FUNCTION_BLOCK FB_Reactor_Set
VAR_IN_OUT
	//stop_reactor_set													: BOOL;
	stop_rs_automode													: BOOL;
	clear_reactor_set_pause												: BOOL;
END_VAR
VAR_INPUT
	r1																	: FB_Reactor;
	
	rs_name																: STRING;
	cycle_mode															: STRING;
//	stop_rs_automode													: BOOL;
	clear_rs_pause														: BOOL;
	open_doors															: BOOL;
	close_doors															: BOOL;
	close_valves														: BOOL;
	retract_clamps														: BOOL;
	extend_clamps														: BOOL;
	
	{attribute 'OPC.UA.DA' := '1'}  				                
	fan_setpoint														: REAL;
	{attribute 'OPC.UA.DA' := '1'}  				                
	{attribute 'OPC.UA.DA.Access' := '1'}  				                
	ti_Cycle_Count														: INT; 
	{attribute 'OPC.UA.DA' := '1'}  				                
	{attribute 'OPC.UA.DA.Access' := '1'}  				                
	ti_Total_Cycle_Count												: DINT; 
	{attribute 'OPC.UA.DA' := '1'}  				                
	{attribute 'OPC.UA.DA.Access' := '1'}  				                
	cycle_stage															: STRING;
    /// <summary>RS_XV08</summary>
	{attribute 'OPC.UA.DA' := '1'}  				                
	steam_bypass_valve													: BOOL;
	/// <summary>XV02</summary>
	{attribute 'OPC.UA.DA' := '1'}  	//mm 11/7 to command valve
	repres_valves														: BOOL;
END_VAR
VAR_OUTPUT
	
	inlet_doors_open													: BOOL;
	inlet_doors_closed													: BOOL;
	outlet_doors_open													: BOOL;
	outlet_doors_closed													: BOOL;

	inlet_clamps_extended												: BOOL;
	inlet_clamps_retracted												: BOOL;
	outlet_clamps_extended												: BOOL;
	outlet_clamps_retracted												: BOOL;
	
	rs_valves_clear														: BOOL;
	adsorption_high_temp_count											: INT;
	desorption_high_temp_count											: INT;
	vacuum_cooling_high_temp_count										: INT;
	sorbent_high_temp													: REAL;
	sorbent_average_temp												: REAL;
	
    /// <summary>Reactor XV02</summary>
	repres_valves_clear													: BOOL;
    /// <summary>RS_XV04</summary>
	dead_air_valve_clear												: BOOL;
    /// <summary>RS_XV05</summary>
	product_iso_valve_clear												: BOOL;
    /// <summary>RS_XV06</summary>
	condensate_valve_clear												: BOOL;
    /// <summary>RS_XV07</summary>
	steam_iso_valve_clear												: BOOL;
    /// <summary>RS_XV08</summary>
	steam_bypass_valve_clear											: BOOL;
	
	/// <summary>RS_LS01</summary>
	{attribute 'OPC.UA.DA' := '1'}  				                
	{attribute 'OPC.UA.DA.Access' := '1'}  				                
	reactor_drain_vessel_lsl									AT %I*	: BOOL;
    /// <summary>RS_LS02</summary>
	{attribute 'OPC.UA.DA' := '1'}  				                
	{attribute 'OPC.UA.DA.Access' := '1'}  				                
	reactor_drain_vessel_lsh									AT %I*	: BOOL;

    /// <summary>RS_FT02</summary>
	{attribute 'OPC.UA.DA' := '1'}  				                
	{attribute 'OPC.UA.DA.Access' := '1'}  				                
	reactor_condensate_flow												: REAL;

	Remaining_Time														: REAL;
	Current_Step														: INT;
	Machine_State														: INT;
	Status																: INT;
	Process_Running														: BOOL;
	Pause_Reactor_Set													: BOOL;
	Reactor_Set_Stopped													: BOOL;
	DoorCycle_Running													: BOOL;
	PositivePressure_Running											: BOOL;
	Repressurization_Running											: BOOL;
	Adsorption_Running													: BOOL;
	Evacuation_Running													: BOOL;
	Desorption_Running													: BOOL;
	Bypass_Running														: BOOL;
	Utility_Error														: BOOL;
	Cancel_Reactor_Set													: BOOL;
	Cancel_All_Reactor_Sets												: BOOL;
	Process_Complete													: BOOL;
	Done																: BOOL;
	
END_VAR
VAR
	eState																: E_MachineState;
	i																	: INT;
	iStatePointer														: INT;
	iLength																: INT;
	iStateMode															: ARRAY[0..9] OF INT;
	stop_reactor_set													: BOOL;
	
	sUtilityError														: STRING;
	sReactorError														: STRING;
	sCancelError														: STRING;
	sRetryError															: STRING;
	sError																: STRING;
	sMessage															: STRING;
	sLeakageAcceptable													: STRING;
	sLeakageUnacceptable												: STRING;

	rAveragePressure													: REAL;
	iCount																: INT;
	iVacuumStatus														: INT;
	iError																: INT;
	
	rTime																: REAL;
	rTime1																: REAL;
	rTime2																: REAL;
	rTime3																: REAL;
	rSP1																: REAL;
	rSP2																: REAL;
	rSP3																: REAL;
	rR1SavedPressure													: REAL;
	rR1Leakage															: REAL;
	rIncrementalMove													: REAL;
	rPosition															: REAL;
	rAverageReactorPres													: REAL;
	rReactorLeakTestStartingPressure									: REAL;
	
	tTime																: TIME;
	
	iStep																: INT;
	i2Step																: INT;
	i3Step																: INT;
	i4Step																: INT;
	i5Step																: INT;
	i6Step																: INT;
	i7Step																: INT;
	i8Step																: INT;
	iStartStep															: INT;
	iStatus																: INT;
	iErrorProcess														: INT;
	iR1Leakage															: INT;
	iCycleCount															: INT;
	iMaxSorbentTempErrorCount											: INT;

	bMultiProcess														: BOOL;
	bEndProcess															: BOOL;
	bSPAdjust															: BOOL;
	bPaused																: BOOL;
	bClearingCycle														: BOOL;
	bDoorCycleDone								        				: BOOL;
	bPositivePressureDone						        				: BOOL;
	bRepressurizationDone												: BOOL;
	bAdsorptionDone														: BOOL;
	bEvacuationDone														: BOOL;
	bDesorptionDone									        			: BOOL;
	bBypassDone									        				: BOOL;
	bPass1																: BOOL;
	bPass2																: BOOL;
	bPass3																: BOOL;
	bPass4																: BOOL;
	bPass5																: BOOL;
	bPass6																: BOOL;
	bPass7																: BOOL;
	bPass8																: BOOL;
	bPass9																: BOOL;
	bPass10																: BOOL;
	
	
	bCondenserKnockoutOn												: BOOL;
	bStop																: BOOL;
	bTimer1																: BOOL;
	bTimer2																: BOOL;
	bTimer3																: BOOL;
	bRunning															: BOOL;
	bDrainError															: BOOL;
	bPumpOn																: BOOL;
	bPumpTimeOut														: BOOL;									
	bDrainResetToLSL													: BOOL;
	bProcessStarted														: BOOL;
	bDesorptionErrorCheck												: BOOL;
	bSafeShutdownOn														: BOOL;
	bInletClampsRetracted												: BOOL;
	bInletClampsExtended												: BOOL;
	bOutletClampsRetracted												: BOOL;
	bOutletClampsExtended												: BOOL;
	bVacuumHolding														: BOOL;
	bCondition21														: BOOL;
	bCondition22														: BOOL;
	bCondition11														: BOOL;
	bCondition12														: BOOL;
	
	rtrigStart															: R_TRIG;
	rtrigPaused															: R_TRIG;
	rtrigIdle															: R_TRIG;
	rtrigDoorCycle														: R_TRIG;
	rtrigPositivePressure												: R_TRIG;
	rtrigRepressurization												: R_TRIG;
	rtrigAdsorption														: R_TRIG;
	rtrigEvacuation														: R_TRIG;
	rtrigDesorption														: R_TRIG;
	rtrigBypass															: R_TRIG;
	rtrigSingleProcessAuto												: R_TRIG;
	rtrigDrainLSHOn														: R_TRIG;
	
	tonTimer1															: TON;
	tonTimer2															: TON;
	tonTimer3															: TON;
	tonPause															: TON;
	tonDrain															: TON;
	rtrigCondensateValveOff_DrainOff									: R_TRIG;
	tonProcess															: TON;
	
	tRestartTime														: TIME;

	bSteamHeaderValve													: BOOL;
	bCondition1															: BOOL;
	bCondition2															: BOOL;
	bCondition3															: BOOL;
	
	reactor_drain_adsorption_on											: BOOL;
	tmrDrainAdsorp														: TON;
	waterscale_desorp													: REAL;
	water_scale_change_oor												: BOOL;
	fb_adsorp_reactor_wastewater											: FB_ChangeOfValue;
	
	
	{attribute 'OPC.UA.DA' := '1'}  				                
	{attribute 'OPC.UA.DA.Access' := '1'}  				                
	ti_Machine_State													: INT;
	{attribute 'OPC.UA.DA' := '1'}  				                
	{attribute 'OPC.UA.DA.Access' := '1'}  				                
	ti_Current_Step														: INT;
	{attribute 'OPC.UA.DA' := '1'}  				                
	{attribute 'OPC.UA.DA.Access' := '1'}  				                
	tb_Process_Running													: BOOL;
	{attribute 'OPC.UA.DA' := '1'}  				                
	{attribute 'OPC.UA.DA.Access' := '1'}  				                
	tb_Repressurization_Running											: BOOL;
	{attribute 'OPC.UA.DA' := '1'}  				                
	{attribute 'OPC.UA.DA.Access' := '1'}  				                
	tb_Adsorption_Running												: BOOL;
	{attribute 'OPC.UA.DA' := '1'}  				                
	{attribute 'OPC.UA.DA.Access' := '1'}  				                
	tb_Evacuation_Running												: BOOL;
	{attribute 'OPC.UA.DA' := '1'}  				                
	{attribute 'OPC.UA.DA.Access' := '1'}  				                
	tb_Desorption_Running												: BOOL;
	{attribute 'OPC.UA.DA' := '1'}  				                
	{attribute 'OPC.UA.DA.Access' := '1'}  				                
	tb_Bypass_Running													: BOOL;
	{attribute 'OPC.UA.DA' := '1'}  				                
	{attribute 'OPC.UA.DA.Access' := '1'}  				                
	tb_Process_Complete													: BOOL;
	{attribute 'OPC.UA.DA' := '1'}  				                
	{attribute 'OPC.UA.DA.Access' := '1'}  				                
	tr_Remaining_Time													: REAL;
	{attribute 'OPC.UA.DA' := '1'}  				                
	{attribute 'OPC.UA.DA.Access' := '1'}  				                
	ti_Status															: INT;
	{attribute 'OPC.UA.DA' := '1'}  				                
	{attribute 'OPC.UA.DA.Access' := '1'}  				                
	ts_Status_Text														: STRING;		

	

	{attribute 'OPC.UA.DA' := '1'}  				                
	{attribute 'OPC.UA.DA.Access' := '1'}  				                
	interlock_inlet_door_clamps_or										: BOOL;

	{attribute 'OPC.UA.DA' := '1'}  				                
	{attribute 'OPC.UA.DA.Access' := '1'}  				                
	interlock_outlet_door_clamps_or										: BOOL;

	{attribute 'OPC.UA.DA' := '1'}  				                
	interlock_inlet_door_or												: BOOL;
	{attribute 'OPC.UA.DA' := '1'} 		      
	{attribute 'OPC.UA.DA.Access' := '1'}  				                
	interlock_inlet_door_or_status										: BOOL;
	{attribute 'OPC.UA.DA' := '1'}  				                
	{attribute 'OPC.UA.DA.Access' := '1'}  				                
	interlock_outlet_door_or											: BOOL;
	{attribute 'OPC.UA.DA' := '1'}  				                
	{attribute 'OPC.UA.DA.Access' := '1'}  				                
	interlock_outlet_door_or_status										: BOOL;
	
	{attribute 'OPC.UA.DA' := '1'}  				                
	interlock_inlet_door_clamp_or										: BOOL;
	{attribute 'OPC.UA.DA' := '1'}  				                
	{attribute 'OPC.UA.DA.Access' := '1'}  				                
	interlock_inlet_door_clamp_or_status								: BOOL;
	{attribute 'OPC.UA.DA' := '1'}  						                
	interlock_outlet_door_clamp_or										: BOOL;
	{attribute 'OPC.UA.DA' := '1'}  				                
	{attribute 'OPC.UA.DA.Access' := '1'}  				                
	interlock_outlet_door_clamp_or_status								: BOOL;
	
    /// <summary>PWR-01</summary>
	{attribute 'OPC.UA.DA' := '1'}  				                
	power_control														: BOOL;
    /// <summary>PWR-01</summary>
	{attribute 'OPC.UA.DA' := '1'}  				                
	{attribute 'OPC.UA.DA.Access' := '1'}  				                
	power_control_status												: BOOL;
    /// <summary>power_cmd</summary>
	PWR_01														AT %Q*	: BOOL;
	circuit_breaker_no_feedback									AT %I*	: BOOL;
	circuit_breaker_nc_feedback									AT %I*	: BOOL;
	

    /// <summary>RS_TT01</summary>
	{attribute 'OPC.UA.DA' := '1'}  				                
	{attribute 'OPC.UA.DA.Access' := '1'}  				                
	product_line_temp													: REAL;
    /// <summary>RS_TT01</summary>
	{attribute 'OPC.UA.DA' := '1'}  				                
	{attribute 'OPC.UA.DA.Access' := '1'}
	product_line_temp_error												: BOOL;
    /// <summary>RS_TT01</summary>
	{attribute 'OPC.UA.DA' := '1'}  				                
	_ProductLineTempErrorOff											: BOOL		:= TRUE;
    /// <summary>rs product line temp</summary>
	TT_01														AT %I*	: INT;
    /// <summary>rs product line temp</summary>
	TT_01_error													AT %I*	: BOOL;
	
    /// <summary>RS_PT02</summary>
	{attribute 'OPC.UA.DA' := '1'}  				                
	{attribute 'OPC.UA.DA.Access' := '1'}  				                
	product_line_pres													: REAL;
    /// <summary>RS_PT02</summary>
	{attribute 'OPC.UA.DA' := '1'}  				                
	{attribute 'OPC.UA.DA.Access' := '1'}  				                
	product_line_pres_error												: BOOL;
    /// <summary>RS_PT02</summary>
	{attribute 'OPC.UA.DA' := '1'}  				                
	_ProductLinePresErrorOff											: BOOL;
    /// <summary>rs product line temp</summary>
	PT_02														AT %I*	: INT;
    /// <summary>rs product line temp</summary>
	PT_02_error													AT %I*	: BOOL;
	
    /// <summary>RS_FT02</summary>
	{attribute 'OPC.UA.DA' := '1'}  				                
	{attribute 'OPC.UA.DA.Access' := '1'}  				                
	reactor_condensate_flow_error										: BOOL;
    /// <summary>RS_FT02</summary>
	{attribute 'OPC.UA.DA' := '1'}  				                
	_ReactorCondensateFlowErrorOff										: BOOL;
    /// <summary>rs reactor condensate flow</summary>
	FT_02														AT %I*	: INT;
    /// <summary>rs reactor condensate flow</summary>
	FT_02_error													AT %I*	: BOOL;

    /// <summary>RS_XV04</summary>
	{attribute 'OPC.UA.DA' := '1'}  				                
	dead_air_valve														: BOOL;
    /// <summary>RS_XV04</summary>
	{attribute 'OPC.UA.DA' := '1'}  				                
	{attribute 'OPC.UA.DA.Access' := '1'}  				                
	dead_air_valve_open_cmd_status										: BOOL;
    /// <summary>RS_XV04</summary>
	{attribute 'OPC.UA.DA' := '1'}  				                
	{attribute 'OPC.UA.DA.Access' := '1'}  				                
	dead_air_valve_open											AT %I*	: BOOL;
    /// <summary>RS_XV04</summary>
	{attribute 'OPC.UA.DA' := '1'}  				                
	{attribute 'OPC.UA.DA.Access' := '1'}  				                
	dead_air_valve_closed										AT %I*	: BOOL;
    /// <summary>dead air valve</summary>
	XV_04														AT %Q*	: BOOL;
	
    /// <summary>RS_XV05</summary>
	{attribute 'OPC.UA.DA' := '1'}  				                
	product_iso_valve													: BOOL;
    /// <summary>RS_XV05</summary>
	{attribute 'OPC.UA.DA' := '1'}  				                
	{attribute 'OPC.UA.DA.Access' := '1'}  				                
	product_iso_valve_open_cmd_status									: BOOL;
    /// <summary>RS_XV05</summary>
	{attribute 'OPC.UA.DA' := '1'}  				                
	{attribute 'OPC.UA.DA.Access' := '1'}  				                
	product_iso_valve_open										AT %I*	: BOOL;
    /// <summary>RS_XV05</summary>
	{attribute 'OPC.UA.DA' := '1'}  				                
	{attribute 'OPC.UA.DA.Access' := '1'}  				               
	product_iso_valve_closed									AT %I*	: BOOL;
    /// <summary>rs product iso valve</summary>
	XV_05														AT %Q*	: BOOL;
	
     /// <summary>RS_XV06</summary>
	{attribute 'OPC.UA.DA' := '1'}  				                
	condensate_valve													: BOOL;
    /// <summary>RS_XV06</summary>
	{attribute 'OPC.UA.DA' := '1'}  				                
	{attribute 'OPC.UA.DA.Access' := '1'}  				                
	condensate_valve_open_cmd_status									: BOOL;
    /// <summary>RS_XV06</summary>
	{attribute 'OPC.UA.DA' := '1'}  				                
	{attribute 'OPC.UA.DA.Access' := '1'}  				                
	condensate_valve_open										AT %I*	: BOOL;
    /// <summary>RS_XV06</summary>
	{attribute 'OPC.UA.DA' := '1'}  				                
	{attribute 'OPC.UA.DA.Access' := '1'}  				                
	condensate_valve_closed										AT %I*	: BOOL;
    /// <summary>cooling valve</summary>
	XV_06														AT %Q*	: BOOL;
	
    /// <summary>RS_XV07</summary>
	{attribute 'OPC.UA.DA' := '1'}  				                
	steam_iso_valve														: BOOL;
    /// <summary>RS_XV07</summary>
	{attribute 'OPC.UA.DA' := '1'}  				                
	{attribute 'OPC.UA.DA.Access' := '1'}  				                
	steam_iso_valve_open_cmd_status										: BOOL;
    /// <summary>RS_XV07</summary>
	{attribute 'OPC.UA.DA' := '1'}  				                
	{attribute 'OPC.UA.DA.Access' := '1'}  				                
	steam_iso_valve_closed										AT %I*	: BOOL;
    /// <summary>RS_XV07</summary>
	{attribute 'OPC.UA.DA' := '1'}  				                
	{attribute 'OPC.UA.DA.Access' := '1'}  				                
	steam_iso_valve_open										AT %I*	: BOOL;
    /// <summary>steam isolation valve</summary>
	XV_07														AT %Q*	: BOOL;

    /// <summary>RS_XV08</summary>
	{attribute 'OPC.UA.DA' := '1'}  				                
	{attribute 'OPC.UA.DA.Access' := '1'}  				                
	steam_bypass_valve_open_cmd_status									: BOOL;
    /// <summary>RS_XV08</summary>
	{attribute 'OPC.UA.DA' := '1'}  				                
	{attribute 'OPC.UA.DA.Access' := '1'}  				                
	steam_bypass_valve_open										AT %I*	: BOOL;
    /// <summary>RS_XV08</summary>
	{attribute 'OPC.UA.DA' := '1'}  				                
	{attribute 'OPC.UA.DA.Access' := '1'}  				                
	steam_bypass_valve_closed									AT %I*	: BOOL;
    /// <summary>steam bypass valve</summary>
	XV_08														AT %Q*	: BOOL;

	{attribute 'OPC.UA.DA' := '1'}  				                
	{attribute 'OPC.UA.DA.Access' := '1'}  				                
	reactor_test_leakage_pressure										: REAL;

END_VAR
VAR PERSISTENT
	
	{attribute 'OPC.UA.DA' := '1'}
	SP_include_inlet_doors_in_process									: BOOL;					
	{attribute 'OPC.UA.DA' := '1'}
	SP_include_outlet_doors_in_process									: BOOL;					

    /// <summary>TT01</summary>
	{attribute 'OPC.UA.DA' := '1'}  				                
	product_line_temp_offset											: REAL;

    /// <summary>PT02</summary>
	{attribute 'OPC.UA.DA' := '1'}  				                
	product_line_pres_low												: REAL;
    /// <summary>PT02</summary>
	{attribute 'OPC.UA.DA' := '1'}  				                
	product_line_pres_high												: REAL;
    /// <summary>PT02</summary>
	{attribute 'OPC.UA.DA' := '1'}  				                
	product_line_pres_min												: REAL;
    /// <summary>PT02</summary>
	{attribute 'OPC.UA.DA' := '1'}  				                
	product_line_pres_offset											: REAL;
	
    /// <summary>RS FT02</summary>
	{attribute 'OPC.UA.DA' := '1'}  				                
	reactor_condensate_flow_low											: REAL;
    /// <summary>RS FT02</summary>
	{attribute 'OPC.UA.DA' := '1'}  				                
	reactor_condensate_flow_high										: REAL;
    /// <summary>RS FT02</summary>
	{attribute 'OPC.UA.DA' := '1'}  				                
	reactor_condensate_flow_min											: REAL;
    /// <summary>RS FT02</summary>
	{attribute 'OPC.UA.DA' := '1'}  				                
	reactor_condensate_flow_offset										: REAL;
	
END_VAR

// Theseus - FB_Reactor_Set
// Rev 1.0 - December 2, 2024

r1(unit := 1);

A_Reactor_Set_IO();

IF eState <> eIdle THEN 
	A_Clear_Variables();
END_IF

iLength																	:= LEN(cycle_mode);
rtrigStart(CLK:= iLength > 0);
IF rtrigStart.Q THEN
	IF cycle_mode = '0' THEN
		bClearingCycle													:= TRUE;											// This acts as if the cycle ran so the reactor set cycle counter will stay in sync with the other reactor sets		
	ELSE
		bProcessStarted													:= TRUE;
		IF Pause_Reactor_Set THEN
			bPaused														:= TRUE;
		ELSE
			iStartStep													:= 1;
			Process_Running												:= TRUE;
			bMultiProcess												:= iLength > 1;
			giEvacuationCounter											:= 0;
			FOR i := 1 TO iLENGTH DO
				iStateMode[i]											:= STRING_TO_INT(MID(cycle_mode, 1, i));
				IF (iStateMode[i] = 6) THEN
					gbFirstEvacuation									:= TRUE;
					giEvacuationCounter									:= giEvacuationCounter + 1;
				END_IF
			END_FOR
			iStatePointer												:= 1;
			Machine_State												:= iStateMode[1];
		END_IF
	END_IF
END_IF

rtrigIdle(				CLK:= eState <= eIdle);
rtrigPaused(			CLk:= bPaused);
rtrigDoorCycle(			CLK:= Machine_State = eDoorCycle);
rtrigSingleProcessAuto(	CLK:= Machine_State = eSingleProcessAuto);
rtrigRepressurization(	CLK:= Machine_State = eRepressurization);
rtrigAdsorption(		CLK:= Machine_State = eAdsorption);
rtrigEvacuation(		CLK:= Machine_State = eEvacuation);
rtrigPositivePressure(	CLK:= Machine_State = ePositivePressure);
rtrigDesorption(		CLK:= Machine_State = eDesorption);
rtrigBypass(			CLK:= Machine_State = eBypass);

IF rtrigPaused.Q THEN
	bPaused																:= FALSE;
	eState																:= ePause;
ELSIF rtrigDoorCycle.Q THEN
	bDoorCycleDone														:= FALSE;
	i2Step																:= iStartStep;
	eState																:= eDoorCycle;
ELSIF rtrigPositivePressure.Q THEN
	bPositivePressureDone												:= FALSE;
	i3Step																:= iStartStep;
	eState																:= ePositivePressure;
ELSIF rtrigRepressurization.Q THEN
	bRepressurizationDone												:= FALSE;
	i4Step																:= iStartStep;
	eState																:= eRepressurization;
ELSIF rtrigAdsorption.Q THEN
	bAdsorptionDone														:= FALSE;
	i5Step																:= iStartStep;
	eState																:= eAdsorption;
ELSIF rtrigEvacuation.Q THEN
	bEvacuationDone														:= FALSE;
	i6Step																:= iStartStep;
	eState																:= eEvacuation;
ELSIF rtrigDesorption.Q THEN
	bDesorptionDone														:= FALSE;
	i7Step																:= iStartStep;
	eState																:= eDesorption;
ELSIF rtrigBypass.Q THEN
	bBypassDone															:= FALSE;
	i8Step																:= iStartStep;
	eState																:= eBypass;
ELSIF rtrigSingleProcessAuto.Q THEN
	eState																:= eSingleProcessAuto;
ELSIF rtrigIdle.Q THEN
	bProcessStarted														:= FALSE;
	eState																:= eIdle;
END_IF

CASE eState OF
	
	eIdle:
		A_Idle();
		
	eDoorCycle:
		IF bDoorCycleDone THEN
			DoorCycle_Running											:= FALSE;
			IF bMultiProcess THEN
				eState													:= SEL(bStop, eChangeState, ePause);
			ELSE
				Status													:= SEL(bStop, eDoorCycle_Complete, Status);
				eState													:= ePause;
			END_IF
		ELSIF bStop THEN
			Status														:= eStopping_Process;
		ELSE
			Status														:= eDoorCycle_Running;
			DoorCycle_Running											:= TRUE;
		END_IF
		
	ePositivePressure:
		IF bPositivePressureDone THEN
			PositivePressure_Running									:= FALSE;
			IF bMultiProcess THEN
				eState													:= SEL(bStop, eChangeState, ePause);
			ELSE
				Status													:= SEL(bStop, ePositivePressure_Complete, Status);
				eState													:= ePause;
			END_IF
		ELSIF bStop THEN
			Status														:= eStopping_Process;
		ELSE
			Status														:= ePositivePressure_Running;
			PositivePressure_Running									:= TRUE;
		END_IF

	eRepressurization:
		IF bRepressurizationDone THEN
			Repressurization_Running									:= FALSE;
			IF bMultiProcess THEN
				eState													:= SEL(bStop, eChangeState, ePause);
			ELSE
				Status													:= SEL(bStop, eRepressurization_Complete, Status);
				eState													:= ePause;
			END_IF
		ELSIF bStop THEN
			Status														:= eStopping_Process;
		ELSE
			Status														:= eRepressurization_Running;
			Repressurization_Running									:= TRUE;
		END_IF

	eAdsorption:
		IF bAdsorptionDone THEN
			Adsorption_Running											:= FALSE;
			IF bMultiProcess THEN
				eState													:= SEL(bStop, eChangeState, ePause);
			ELSE
				Status													:= SEL(bStop, eAdsorption_Complete, Status);
				eState													:= ePause;
			END_IF
		ELSIF bStop THEN
			Status														:= eStopping_Process;
		ELSE
			Status														:= eAdsorption_Running;
			Adsorption_Running											:= TRUE;
		END_IF

	eEvacuation:
		IF bEvacuationDone THEN
			Evacuation_Running											:= FALSE;
			IF bMultiProcess THEN
				eState													:= SEL(bStop, eChangeState, ePause);
			ELSE
				Status													:= SEL(bStop, eEvacuation_Complete, Status);
				eState													:= ePause;
			END_IF
		ELSIF bStop THEN
			Status														:= eStopping_Process;
		ELSE
			Status														:= eEvacuation_Running;
			Evacuation_Running											:= TRUE;
		END_IF
		
	eDesorption:
		IF bDesorptionDone THEN
			Desorption_Running											:= FALSE;
			IF bMultiProcess THEN
				eState													:= SEL(bStop, eChangeState, ePause);
			ELSE
				Status													:= SEL(bStop, eDesorption_Complete, Status);
				eState													:= ePause;
			END_IF
		ELSIF bStop THEN
			Status														:= eStopping_Process;
		ELSE
			Status														:= eDesorption_Running;
			Desorption_Running											:= TRUE;
		END_IF
		
	eBypass:
		IF bBypassDone THEN
			Bypass_Running												:= FALSE;
			IF bMultiProcess THEN
				eState													:= SEL(bStop, eChangeState, ePause);
			ELSE
				Status													:= SEL(bStop, eBypass_Complete, Status);
				eState													:= ePause;
			END_IF
		ELSIF bStop THEN
			Status														:= eStopping_Process;
		ELSE
			Status														:= eBypass_Running;
			Bypass_Running												:= TRUE;
		END_IF
		
	eSingleProcessAuto:
		eState															:= eChangeState;
		
	eChangeState:
		iStatePointer													:= iStatePointer + 1;
		IF iStatePointer > iLength THEN
			Process_Complete											:= TRUE;
			Done														:= TRUE;
			eState														:= eIdle;
		ELSIF iStateMode[iStatePointer] = 0 THEN
			Status														:= eStopping_Process;
			bStop														:= TRUE;
			bMultiProcess												:= FALSE;
			eState														:= ePause;
		ELSE
			Machine_State												:= iStateMode[iStatePointer];
		END_IF
	
	ePause:
		Machine_State													:= ePause;
		IF tonPause.Q THEN
			Done														:= TRUE;
			eState														:= eIdle;
		END_IF
		
END_CASE

bRunning																:= eState >= eRepressurization AND eState <= ePause;

A2_DoorCycle_1();
A3_PositivePressure_1();
A4_Repressurization_1();
A5_Adsorption_1();
A6_Evacuation_1();
A7_Desorption_1();
A8_Bypass_1();

(*
A4_Repressurization();
A5_Adsorption();
A6_Evacuation();
A7_Desorption();
A8_Bypass();
*)


A_Drain_Reactor_Set();

tonTimer1(IN:= bTimer1, PT:= REAL_TO_TIME(rTime1));
tonTimer2(IN:= bTimer2, PT:= REAL_TO_TIME(rTime2));
tonTimer3(IN:= bTimer3, PT:= REAL_TO_TIME(rTime3));

Remaining_Time															:= 0;
IF Process_Running THEN
	IF bTimer1 THEN
		Remaining_Time													:= rTime1 - TIME_TO_REAL(tonTimer1.ET);
	ELSIF bTimer2 THEN
		Remaining_Time													:= rTime2 - TIME_TO_REAL(tonTimer2.ET);
	ELSIF bTimer3 THEN
		Remaining_Time													:= rTime3 - TIME_TO_REAL(tonTimer3.ET);
	END_IF
END_IF

tonPause(IN:= eState = ePause, PT:= _TIMEOUT_RESET);
tonProcess(IN:= bProcessStarted, PT:= T#10H);

ti_Current_Step := Current_Step;
tr_Remaining_Time := Remaining_Time;
tb_Process_Running := Process_Running;

ACTION A_Check_Process:
// Theseus - FB_Reactor_Set.A_ClearProcess
// Rev 1.0 - June 13, 2024

Current_Step															:= iStep;
bEndProcess																:= FALSE;
IF stop_reactor_set THEN																									// Reactor Set can be stopped both internally and externally
	stop_reactor_set													:= FALSE;											// Clear flag
	bEndProcess															:= TRUE;											// Set flag to end process
ELSE
	IF sUtilityError <> '' THEN
		sError															:= sUtilityError;
		Utility_Error													:= TRUE;
		iStep															:= 98;
	ELSIF sReactorError <> '' THEN
		sError															:= sReactorError;
  		bEndProcess														:= TRUE;
	END_IF
	IF sError <> '' THEN
		P_Alarms.M_Add_Alarm(rs_name, F_Concat3(cycle_stage, ' ', sError), sMessage);
		sError															:= '';
	END_IF
END_IF

IF bEndProcess THEN
	bTimer1								 								:= FALSE;
	bTimer2								 								:= FALSE;
	bStop																:= TRUE;
	iStep																:= SEL(bMultiProcess, 80, 90);
END_IF
END_ACTION

ACTION A_Clear_Variables:
// Theseus - FB_Reactor_Set.A_Clear_Variables
// Rev 1.0 - November 26, 2024

//close_all_valves													:= FALSE;
//co2_sensors_on														:= FALSE;
Utility_Error															:= FALSE;
Cancel_Reactor_Set														:= FALSE;
Cancel_All_Reactor_Sets													:= FALSE;
sUtilityError															:= '';
sReactorError															:= '';
sRetryError																:= '';
IF clear_reactor_set_pause THEN
	clear_reactor_set_pause												:= FALSE;
	Pause_Reactor_Set													:= FALSE;
END_IF
IF NOT P_U01.auto_mode_on THEN
	iMaxSorbentTempErrorCount											:= 0;
	iCycleCount															:= 0;	
END_IF
END_ACTION

ACTION A_Drain_Reactor_Set:
// Theseus - FB_Reactor_Set.A_Drain_Reactor_Set
// Rev 1.0 - October 4, 2024

IF (gbDrainageOn OR P_U01.reactor_drain_or_on) AND NOT P_U01.reactor_drain_or_off THEN
	IF NOT r1.reactor_pres_error AND r1.reactor_pres >= P_U01.SP_minimum_drainage_pressure THEN
//		tonDrain(IN:= NOT bDrainError AND condensate_valve, PT:= REAL_TO_TIME(P_U01.SP_maximum_duration_to_drain_reactor_set * _SECONDS));
		IF tonDrain.Q AND reactor_condensate_flow < P_U01.SP_minimum_condensate_flow THEN
			condensate_valve											:= FALSE;
			IF TRUE THEN ///@@@reactor_drain_vessel_high THEN
				P_U01.steam_flow_control_valve							:= _CLOSED;
				P_Alarms.M_Add_Alarm(rs_name, gsReactorDrainError, gsMessageTBD);
				bDrainError												:= TRUE;
			END_IF
		ELSIF reactor_drain_vessel_lsh THEN ///@@@reactor_drain_vessel_high THEN							mm 11/7 
			condensate_valve											:= TRUE;
		ELSIF NOT reactor_drain_vessel_lsh AND NOT reactor_drain_vessel_lsl THEN ///@@@reactor_drain_vessel_low AND NOT reactor_drain_vessel_high THEN
			condensate_valve											:= FALSE;
//			bDrainError													:= FALSE;
		END_IF
	ELSE
//		IF NOT P_U01.reactor_drain_or_off  THEN 
			condensate_valve												:= FALSE;
//		END_IF
	END_IF
END_IF

rtrigCondensateValveOff_DrainOff(CLK := NOT gbDrainageOn AND NOT P_U01.reactor_drain_or_on AND NOT P_U01.reactor_drain_or_off);
IF 	rtrigCondensateValveOff_DrainOff.Q THEN
	condensate_valve												:= FALSE;
END_IF


gbCondensateValve														:= condensate_valve;

fb_adsorp_reactor_wastewater
	( i_execute := reactor_drain_adsorption_on,
	  i_value := P_U01.water_scale_3,
	  i_time := 30,
	  i_threshold := 1);
	  
IF reactor_drain_adsorption_on THEN
	IF NOT fb_adsorp_reactor_wastewater.o_below_threshold THEN
		condensate_valve											:= TRUE;
	ELSIF fb_adsorp_reactor_wastewater.o_below_threshold OR fb_adsorp_reactor_wastewater.o_timeout THEN
		condensate_valve											:= FALSE;
		reactor_drain_adsorption_on := FALSE;
	END_IF
END_IF
END_ACTION

ACTION A_Idle:
// Theseus - FB_Reactor_Set.A_Idle
// Rev 1.0 - June 24, 2024

Machine_State															:= eIdle;
cycle_stage																:= 'idle.idle';
sError																	:= '';
i4Step																	:= 0;
i5Step																	:= 0;
i6Step																	:= 0;
i7Step																	:= 0;
Current_Step															:= 0;
Remaining_Time															:= 0;
Current_Step															:= 0;
Status																	:= 0;
bMultiProcess															:= FALSE;
bTimer1																	:= FALSE;
bTimer2																	:= FALSE;
bStop																	:= FALSE;
Process_Running															:= FALSE;
Process_Complete														:= FALSE;
IF bClearingCycle THEN
	Done																:= TRUE;
	bClearingCycle														:= FALSE;
ELSE
	Done																:= FALSE;
END_IF
END_ACTION

ACTION A_Reactor_Set_IO:
// Theseus - A_Reactor_Set_IO
// Rev 1.0 - November 26, 2024

r1.fan_vfd_setpoint														:= fan_setpoint;

repres_valves_clear														:= r1.repres_valve_clear;

rAverageReactorPres														:= r1.reactor_pres;

//rso_power_control_out													:= rsi_power_control_fdbk_no AND NOT rsi_power_control_fdbk_nc AND NOT rso_PWR_01 ;
//rso_PWR_01																:= rsi_power_control_in;

interlock_inlet_door_or_status											:= interlock_inlet_door_or;
interlock_outlet_door_or_status											:= interlock_outlet_door_or;
interlock_inlet_door_clamp_or_status									:= interlock_inlet_door_clamp_or;
interlock_outlet_door_clamp_or_status									:= interlock_outlet_door_clamp_or;

inlet_doors_open														:= r1.inlet_doors_open;
inlet_doors_closed														:= r1.inlet_doors_closed;
outlet_doors_open														:= r1.outlet_doors_open;
outlet_doors_closed			 											:= r1.outlet_doors_closed;
 
gbGasketsActivated														:= SEL(NOT inlet_doors_closed OR NOT outlet_doors_closed, gbGasketsActivated, FALSE);					// PS 08_20_24

inlet_clamps_extended													:= r1.inlet_door_clamps_extended;
inlet_clamps_retracted													:= r1.inlet_door_clamps_retracted;
outlet_clamps_extended													:= r1.outlet_door_clamps_extended;
outlet_clamps_retracted													:= r1.outlet_door_clamps_retracted;

IF close_valves THEN
	dead_air_valve														:= FALSE;
	product_iso_valve													:= FALSE;
	condensate_valve													:= FALSE;
	steam_iso_valve														:= FALSE;
	steam_bypass_valve													:= FALSE;
	close_valves														:= FALSE;
END_IF

// Interlock 12
P_U01.door_open_with_steam_flow_interlock								:= NOT P_U01.steam_flow_control_valve_closed AND NOT steam_iso_valve_closed;
bCondition21															:= NOT P_U01.interlock_door_open_with_steam_flow_or AND P_U01.door_open_with_steam_flow_interlock;

// Interlock 14
P_U01.door_open_with_reactor_vacuum_interlock							:= rAverageReactorPres < 0.95;
bCondition22															:= NOT P_U01.interlock_door_open_with_reactor_vacuum_or AND P_U01.door_open_with_reactor_vacuum_interlock;

IF open_doors THEN
	r1.open_inlet_door													:= (inlet_clamps_retracted OR interlock_inlet_door_clamp_or)  AND NOT bCondition21 AND NOT bCondition22; // AND SP_include_inlet_doors_in_process;
	r1.open_outlet_door													:= (outlet_clamps_retracted OR interlock_outlet_door_clamp_or)  AND NOT bCondition21 AND NOT bCondition22; // AND SP_include_outlet_doors_in_process;
	open_doors															:= FALSE;
END_IF
IF close_doors THEN
	r1.close_inlet_door													:= (inlet_clamps_retracted OR interlock_inlet_door_clamp_or) ; //AND SP_include_inlet_doors_in_process;
	r1.close_outlet_door												:= (outlet_clamps_retracted OR interlock_outlet_door_clamp_or); // AND SP_include_outlet_doors_in_process;
	close_doors															:= FALSE;
END_IF

IF extend_clamps THEN
	r1.extend_inlet_door_clamps											:= (inlet_doors_closed OR interlock_inlet_door_or) AND SP_include_inlet_doors_in_process;
	r1.extend_outlet_door_clamps										:= (outlet_doors_closed OR interlock_outlet_door_or) AND SP_include_outlet_doors_in_process;
	extend_clamps														:= FALSE;
END_IF
IF retract_clamps THEN
	r1.retract_inlet_door_clamps										:= SP_include_inlet_doors_in_process;
	r1.retract_outlet_door_clamps										:= SP_include_outlet_doors_in_process;
	retract_clamps														:= FALSE;
END_IF

// CO2 adsorption sensor function
P_U01.co2_adsorption_interlock											:= r1.fan_vfd_setpoint > 10 AND r1.sorbent_high_temp < P_M01.SP_maximum_safe_co2_adsorption_sensor_temperature;
IF NOT P_U01.interlock_co2_adsorption_or THEN
	r1.inlet_co2_sol													:= P_U01.co2_adsorption_interlock;
	r1.outlet_co2_sol													:= P_U01.co2_adsorption_interlock;
	r1.outlet_co2_pump													:= TRUE;
	r1.inlet_co2_pump													:= TRUE;
ELSE
	r1.outlet_co2_pump													:= FALSE;
	r1.inlet_co2_pump													:= FALSE;
END_IF


r1.repres_valve															:= repres_valves AND gbRepresValves;

// Interlock 3
P_U01.hot_reactor_condenser_interlock									:= r1.temp_average > P_M01.SP_maximum_sorbent_temperature_to_use_dead_air_line;
IF NOT P_U01.interlock_hot_reactor_condenser_or and P_U01.hot_reactor_condenser_interlock THEN
	dead_air_valve														:= FALSE;
END_IF

XV_04																	:= dead_air_valve;
dead_air_valve_open_cmd_status											:= XV_04;
dead_air_valve_clear													:= F_ValveClear(dead_air_valve, dead_air_valve_open, dead_air_valve_closed);

XV_05																	:= product_iso_valve;
product_iso_valve_open_cmd_status										:= XV_05;
product_iso_valve_clear													:= F_ValveClear(product_iso_valve, product_iso_valve_open, product_iso_valve_closed);

XV_06																	:= condensate_valve;
condensate_valve_open_cmd_status										:= XV_06;
condensate_valve_clear													:= F_ValveClear(condensate_valve, condensate_valve_open, condensate_valve_closed);

// Interlock 4
P_U01.no_steam_unevacuated_reactor_interlock							:= r1.temp_high < P_M01.SP_maximum_safe_ambient_temperature AND NOT P_U01.steam_flow_control_valve_closed AND r1.reactor_pres < P_M01.SP_maximum_reactor_pressure_to_introduce_steam;
bCondition1																:= P_U01.interlock_no_steam_unevacuated_reactor_or OR P_U01.no_steam_unevacuated_reactor_interlock;

// Interlock 10
P_U01.reactor_over_safe_pressure_limit_interlock						:= r1.reactor_pres <= P_M01.SP_maximum_safe_reactor_steam_pressure;
bCondition2																:= P_U01.interlock_reactor_over_safe_pressure_limit_or OR P_U01.reactor_over_safe_pressure_limit_interlock;
r1.over_pressure_test_control											:= SEL(NOT bCondition2, r1.over_pressure_test_control, FALSE);

// Interlock 11
P_U01.reactor_over_safe_temperature_limit_interlock						:= r1.temp_high <= P_M01.SP_maximum_safe_sorbent_temperature;
bCondition3																:= P_U01.interlock_reactor_over_safe_temperature_limit_or OR P_U01.reactor_over_safe_temperature_limit_interlock;

IF NOT bCondition1 OR NOT bCondition2 OR NOT bCondition3 THEN
	steam_iso_valve														:= FALSE;
END_IF

XV_07																	:= steam_iso_valve;
steam_iso_valve_open_cmd_status											:= XV_07;
steam_iso_valve_clear													:= F_ValveClear(steam_iso_valve, steam_iso_valve_open, steam_iso_valve_closed);

XV_08																	:= steam_bypass_valve;
steam_bypass_valve_open_cmd_status										:= XV_08;
steam_bypass_valve_clear												:= F_ValveClear(steam_bypass_valve, steam_bypass_valve_open, steam_bypass_valve_closed);

rs_valves_clear															:= dead_air_valve_clear AND product_iso_valve_clear AND steam_iso_valve_clear AND steam_bypass_valve_clear AND condensate_valve_clear;

product_line_temp														:= F_Temperature(TT_01, product_line_temp_offset);
product_line_temp_error													:= TT_01_error AND NOT _ProductLineTempErrorOff;

product_line_pres														:= F_AnalogIn(PT_02, product_line_pres_low, product_line_pres_high, product_line_pres_min, product_line_pres_offset);
product_line_pres_error													:= PT_02_error AND NOT _ProductLinePresErrorOff;

reactor_condensate_flow													:= F_AnalogIn(FT_02, reactor_condensate_flow_low, reactor_condensate_flow_high, reactor_condensate_flow_min, reactor_condensate_flow_offset);
reactor_condensate_flow_error											:= FT_02_error AND NOT _ReactorCondensateFlowErrorOff;


gbCondenserKODrainageOn													:= product_line_pres >= P_U01.SP_minimum_drainage_pressure;

adsorption_high_temp_count												:= r1.adsorption_high_temp_count;
desorption_high_temp_count												:= r1.desorption_high_temp_count;
vacuum_cooling_high_temp_count											:= r1.vacuum_cooling_high_temp_count;
sorbent_high_temp														:= r1.sorbent_high_temp;
sorbent_average_temp													:= r1.sorbent_average_temp;

stop_reactor_set														:= stop_rs_automode;
stop_rs_automode														:= FALSE;
clear_reactor_set_pause													:= clear_rs_pause;
clear_rs_pause															:= FALSE;

//reactor_over_max_pressure												:= NOT r1.reactor_pres_error AND r1.reactor_pres > P_M01.SP_maximum_safe_reactor_steam_pressure;

rAveragePressure														:= 0;
iCount																	:= 0;
iVacuumStatus															:= 0;
iError																	:= 4;
IF NOT r1.reactor_pres_error THEN
	rAveragePressure													:= rAveragePressure + r1.reactor_pres;
	iVacuumStatus														:= F_LowMidHigh(r1.reactor_pres, P_M01.SP_target_desorption_starting_pressure, P_M01.SP_maximum_desorption_starting_pressure, iVacuumStatus);
	iCount																:= iCount + 1;
	iError																:= iError - 1;
END_IF
END_ACTION

ACTION A_Reset:
// Theseus - FB_Reactor_Set.A_Reset
// Rev 1.0 - November 25, 2024

r1.over_pressure_test_control											:= FALSE;
repres_valves															:= FALSE;
//co2_sensors_on														:= FALSE;
dead_air_valve															:= FALSE;
product_iso_valve														:= FALSE;
condensate_valve														:= FALSE;
steam_iso_valve															:= FALSE;
steam_bypass_valve														:= FALSE;
fan_setpoint															:= 0;
END_ACTION

ACTION A2_DoorCycle_1:
// Theseus - FB_Reactor_Set.A2_DoorCycle_1
// Rev 1.0 - June 26, 2024

CASE i2Step OF	

	0:	;
		
	1:
		cycle_stage														:= 'doorcycle.initialize';
		sMessage														:= gsSystemCannotRun;
		rTime1															:= 5 * _SECONDS;
		i2Step															:= i2Step + 1;
		
	2:
		bTimer1															:= TRUE;
		IF tonTimer1.Q THEN
			bTimer1														:= FALSE;
			i2Step														:= 99;
		END_IF
		
	99:
		bDoorCycleDone													:= TRUE;											// 9
		Current_Step													:= 0;
		i2Step															:= 0;
	
	
END_CASE

IF i2Step > 0 AND i2Step < 80 THEN
	iStep																:= i2Step;
	Current_Step														:= iStep;
	A_Check_Process();
	i2Step																:= iStep;
END_IF
END_ACTION

ACTION A2_DoorCycle_OLD:
// Theseus - FB_Reactor_Set.A2_DoorCycle
// Rev 1.0 - October 9, 2024

CASE i2Step OF	

	0:	;
		
	1:
		cycle_stage														:= 'doorcycle.initialize';
		sMessage														:= gsSystemCannotRun;
		IF NOT SP_include_inlet_doors_in_process AND NOT SP_include_outlet_doors_in_process THEN
			sReactorError												:= gsDoorsNotSelectedError;
		ELSIF r1.reactor_pres_error THEN
			sReactorError												:= gsReactorPresSensorError;
		ELSE
			A_Reset();																										// 1
			rTime1														:= 5 * _SECONDS;
			i2Step														:= i2Step + 1;
		END_IF
		
	2:
		bTimer1															:= TRUE;
		IF r1.reactor_pres > 0.98 AND r1.reactor_pres < 1.02 THEN															// 2
			bTimer1														:= FALSE;
			i2Step														:= i2Step + 1;
		ELSIF tonTimer1.Q THEN
			sReactorError												:= gsReactorNotAtAmbientPressure;
		END_IF
		
	3:
		bTimer1															:= TRUE;
		bPass1															:= bInletClampsRetracted;
		bPass2															:= bOutletClampsRetracted;
		IF bPass1 AND bPass2 THEN																							// 3
			bTimer1														:= FALSE;
			repres_valves												:= TRUE;											// 4
			rTime1														:= _VALVE_TIME;
			i2Step														:= i2Step + 1;
		ELSIF tonTimer1.Q THEN
			sReactorError												:= gsClampsNotRetractedError;
		END_IF
	
	4:
		bTimer1															:= TRUE;
		IF repres_valves_clear THEN
			cycle_stage													:= 'doorcycle.open';
			bTimer1														:= FALSE;
			open_doors													:= TRUE;											// 5
			rTime1														:= _DOOR_ACTUATION_TIMEOUT;
			i2Step														:= i2Step + 1;
		ELSIF tonTimer1.Q THEN
			sReactorError												:= gsRepressurizationValveError;
		END_IF
		
	5:
		bTimer1															:= TRUE;
		IF inlet_doors_open AND outlet_doors_open THEN
			bTimer1														:= FALSE;
			rTime1														:= 5 * _SECONDS;
			i2Step														:= i2Step + 1;
		ELSIF tonTimer1.Q THEN
			sReactorError												:= gsInletDoorNotOpenError;
			sReactorError												:= SEL(inlet_doors_open, gsOutletDoorNotOpenError, sReactorError);
		END_IF
		
	6:
		bTimer1															:= TRUE;
		IF tonTimer1.Q THEN																									// 6
			cycle_stage													:= 'doorcycle.close';
			bTimer1														:= FALSE;
			close_doors													:= TRUE;											// 7
			rTime1														:= _DOOR_ACTUATION_TIMEOUT;
			i2Step														:= i2Step + 1;
		END_IF
		
	7:
		bTimer1															:= TRUE;
		IF inlet_doors_closed AND outlet_doors_closed THEN
			bTimer1														:= FALSE;
			rTime1														:= 5 * _SECONDS;
			i2Step														:= i2Step + 1;
		ELSIF tonTimer1.Q THEN
			sReactorError												:= gsInletDoorNotClosedError;
			sReactorError												:= SEL(bPass2, gsOutletDoorNotClosedError, sReactorError);
		END_IF

	8:		
		bTimer1															:= TRUE;
		IF tonTimer1.Q THEN																									// 8
			bTimer1														:= FALSE;
			i2Step														:= 99;
		END_IF
	
	80:																														// Manual process closing
		cycle_stage														:= 'doorcycle.stopping';
		rTime1															:= _STOPPING_TIME;
		A_Reset();
		i2Step															:= 98;
		
	90:																														// Automatic process stopping
		cycle_stage														:= 'doorcycle.stopping';
		rTime1															:= _STOPPING_TIME;
		A_Reset();
		i2Step															:= 98;
		
	98:
		bTimer1															:= TRUE;
		IF tonTimer1.Q THEN
			bTimer1														:= FALSE;
			i2Step														:= 99;
		END_IF
		
	99:
		bDoorCycleDone													:= TRUE;											// 9
		Current_Step													:= 0;
		i2Step															:= 0;
	
	
END_CASE

IF i2Step > 0 AND i2Step < 80 THEN
	iStep																:= i2Step;
	Current_Step														:= iStep;
	A_Check_Process();
	i2Step																:= iStep;
END_IF
END_ACTION

ACTION A3_PositivePressure_1:
// Theseus - FB_Reactor_Set.A3_PositivePressure_1
// Rev 1.0 - June 26, 2024

CASE i3Step OF	

	0:	;
		
	1:
		cycle_stage														:= 'positivepressure.initialize';
		sMessage														:= gsSystemCannotRun;
		rTime1															:= _VALVE_TIME;
		i3Step															:= i3Step + 1;

	2:
		bTimer1															:= TRUE;
		IF tonTimer1.Q THEN
			bTimer1														:= FALSE;
			i3Step														:= 99;
		END_IF
	
	99:
		bPositivePressureDone											:= TRUE;
		Current_Step													:= 0;
		i3Step															:= 0;
	
	
END_CASE

IF i3Step > 0 AND i3Step < 80 THEN
	iStep																:= i3Step;
	Current_Step														:= iStep;
	A_Check_Process();
	i3Step																:= iStep;
END_IF
END_ACTION

ACTION A3_PositivePressure_OLD:
// Theseus - FB_Reactor_Set.A3_PositivePressure
// Rev 1.0 - October 3, 2024

CASE i3Step OF	

	0:	;
		
	1:
		cycle_stage														:= 'positivepressure.initialize';
		sMessage														:= gsSystemCannotRun;
		IF r1.reactor_pres_error THEN
			sReactorError												:= gsReactorPresSensorError;
		ELSE
			A_Reset();																										// 1
			i3Step														:= i3Step + 1;
		END_IF

	2:
		IF gbGasketsActivated THEN																							// 2
			rTime1														:= _VALVE_TIME;
			i3Step														:= i3Step + 1;
		ELSE
			sReactorError												:= gsGasketNotActivatedError;
		END_IF
		
	3:
		bTimer1															:= TRUE;
		IF repres_valves_clear AND rs_valves_clear THEN																	// 3
			bTimer1														:= FALSE;
			i3Step														:= i3Step + 1;
		ELSIF tonTimer1.Q THEN
			sReactorError												:= gsRepressurizationValveError;
			sReactorError												:= SEL(steam_iso_valve_clear, gsSteamIsoValveError, sReactorError);
			sReactorError												:= SEL(steam_bypass_valve_clear, gsSteamBypassValveError, sReactorError);
			sReactorError												:= SEL(product_iso_valve_clear, gsProductIsoValveError, sReactorError);
			sReactorError												:= SEL(dead_air_valve_clear, gsDeadAirValveError, sReactorError);
			sReactorError												:= SEL(condensate_valve_clear, gsCondensateValveError, sReactorError);
		END_IF
	
	4:
		IF bInletClampsExtended AND bOutletClampsExtended THEN																// 4
			cycle_stage													:= 'positivepressure.pressurizing';
			//m01_rs1_r1.XV_09											:= TRUE;											// smrg debug
			r1.over_pressure_test_control								:= TRUE;
			//overpressure_test_control								:= TRUE;											// 5
			rTime1														:= 5 * _MINUTES;
			i3Step														:= i3Step + 1;
		ELSE
			sReactorError												:= gsClampsNotExtendedError;
		END_IF
		
	5:
		bTimer1															:= TRUE;
		IF r1.reactor_pres >= P_M01.SP_pos_pres_ideal_pressure THEN
			bTimer1														:= FALSE;
			cycle_stage													:= 'positivepressure.settling';
			r1.over_pressure_test_control								:= FALSE;											// 6
			rTime1														:= P_M01.SP_pos_pres_settle_time * _MINUTES;		// 7
			i3Step														:= i3Step + 1;
		ELSIF tonTimer1.Q THEN
			sReactorError												:= gsPositivePressureError;
		END_IF
	
	6:
		bTimer1															:= TRUE;
		IF tonTimer1.Q THEN
			rR1SavedPressure											:= r1.reactor_pres;									// 8
			cycle_stage													:= 'positivepressure.leak_test';
			rTime1														:= P_M01.SP_pos_pres_leak_test_duration * _MINUTES;	// 9
			i3Step														:= i3Step + 1;
		END_IF
		
	7:
		bTimer1															:= TRUE;
		IF tonTimer1.Q THEN
			bTimer1														:= FALSE;
			rR1Leakage													:= (r1.reactor_pres - rR1SavedPressure) / P_M01.SP_pos_pres_leak_test_duration;	// 10
			IF rR1Leakage > P_M01.SP_unacceptable_pos_pres_change THEN
				sReactorError											:= gsUnacceptableReactorLeakRate;
			ELSE
				i3Step													:= 99;												// 11
			END_IF
		END_IF
		
	80:																														// Manual process closing
		cycle_stage														:= 'positivePressure.stopping';
		rTime1															:= _STOPPING_TIME;
		A_Reset();
		i3Step															:= 98;
		
	90:																														// Automatic process stopping
		cycle_stage														:= 'positivePressure.stopping';
		rTime1															:= _STOPPING_TIME;
		A_Reset();
		i3Step															:= 98;
		
	98:
		bTimer1															:= TRUE;
		IF tonTimer1.Q THEN
			bTimer1														:= FALSE;
			i3Step														:= 99;
		END_IF
		
	99:
		bPositivePressureDone											:= TRUE;
		Current_Step													:= 0;
		i3Step															:= 0;
	
	
END_CASE

IF i3Step > 0 AND i3Step < 80 THEN
	iStep																:= i3Step;
	Current_Step														:= iStep;
	A_Check_Process();
	i3Step																:= iStep;
END_IF
END_ACTION

ACTION A4_Repressurization:


CASE i4Step OF
	
	0:	;
	
	1: 
		cycle_stage														:= 'repressurization.initialize';
		sMessage														:= gsSystemCannotRun;
		
		IF P_U01.utility_error <> '' THEN
			sUtilityError												:= P_U01.utility_error;
		ELSIF r1.reactor_pres_error THEN
			sReactorError												:= gsReactorPresSensorError;
		ELSE			
//			A_Reset();
			P_U01.boiler_package 										:= FALSE;
			P_U01.steam_flow_control_valve_mode							:= eManual;
			P_U01.steam_flow_control_valve								:= _CLOSED;										
			dead_air_valve												:= FALSE;								// M01.XV04 <- FALSE
			product_iso_valve											:= FALSE;								// M01.XV05 <- FALSE
			steam_bypass_valve											:= FALSE;								// M01.XV08 <- FALSE
			rTime1														:= _VALVE_TIME;			
			i4Step														:= i4Step + 1;												
		END_IF		
		
	2: 
		cycle_stage														:= 'repressurization.starting';	
		bTimer1															:= TRUE;
		bPass1															:= P_U01.steam_flow_control_valve_closed;
		bPass2															:= dead_air_valve_closed;
		bPass3															:= product_iso_valve_clear;
		bPass4															:= steam_bypass_valve_clear;
		IF bPass1 AND bPass2 AND bPass3 AND bPass4  THEN
			bTimer1														:= FALSE; 
			i4Step														:= i4Step + 1;
		ELSIF tonTimer1.Q THEN
			bTimer1														:= FALSE; 
			sUtilityError												:= SEL(bPass1, gsSteamFlowConrolValveError, '');
			sReactorError												:= SEL(bPass2,gsDeadAirValveError,'');
			sReactorError												:= SEL(bPass3, gsProductIsoValveError, sReactorError);
			sReactorError												:= SEL(bPass1,'Steam Bypass Valve Error RS XV08', sReactorError);
		END_IF

	3: 
		bPass1 															:= sorbent_high_temp <= P_M01.SP_maximum_target_sorbent_temperature_to_repressurize;
		bPass2															:= r1.reactor_pres < 0.7;
		IF bPass1 AND bPass2 THEN
			rTime1														:= _CLAMP_ACTUATION_TIMEOUT;
			i4Step														:= i4Step + 1;
			
		ELSE
			sReactorError												:= SEL(bPass1,gsSorbentTemperatureError,'');
			sReactorError												:= SEL(bPass2,gsReactorPressureAboveDesiredLevelError,sReactorError);
		END_IF
		
	4: 
		
		bTimer1															:= TRUE;
		retract_clamps													:= TRUE;
		IF inlet_clamps_retracted AND outlet_clamps_retracted THEN 
			bTimer1														:= FALSE;
			repres_valves												:= TRUE;
			rTime1														:= _VALVE_TIME;
			rTime2														:= 5 * _SECONDS; 
			i4Step														:= i4Step + 1;	
		ELSIF tonTimer1.Q THEN
			bTimer1														:= FALSE; 
			sReactorError												:= gsDoorClampsExtendedError;
		END_IF
		
	5: 
		
		bTimer1															:= TRUE;
		
		IF r1.repres_valve_clear THEN 
			bTimer1														:= FALSE;
			bTimer2														:= TRUE;
			IF tonTimer2.Q THEN 
				bTimer2													:= FALSE;
				steam_iso_valve											:= TRUE;
				rTime1													:= _VALVE_TIME;
				i4Step													:= i4Step + 1;			
			END_IF
		ELSIF tonTimer1.Q THEN
			bTimer1														:= FALSE;
			bTimer2														:= FALSE;
			sReactorError												:= gsRepressurizationValveError;
		END_IF
		
	6: 
		
		bTimer1															:= TRUE;
		
		IF steam_iso_valve_clear THEN
			cycle_stage													:= 'repressurization.repressurize';
			bTimer1														:= FALSE;
			rTime1 														:= 2 * _MINUTES;
			i4Step														:= i4Step + 1;
		ELSIF tonTimer1.Q THEN
			bTimer1														:= FALSE;
			sReactorError												:= gsSteamIsoValveError;
		END_IF
		
	7: 
		
		bTimer1															:= TRUE;
		
		IF r1.reactor_pres > 0.98 AND r1.reactor_pres < 1.02 THEN															
			bTimer1														:= FALSE;
			rTime1														:= 10 * _SECONDS;
			i4Step														:= i4Step + 1;
		ELSIF tonTimer1.Q THEN
			bTimer1														:= FALSE;
			sReactorError												:= gsRepressurizationError;
		END_IF
		
		
	8: 
		
		bTimer1															:= TRUE;
		IF tonTimer1.Q THEN																									
			bTimer1														:= FALSE;
			repres_valves												:= FALSE;
			steam_iso_valve												:= FALSE;
			rTime1														:= _VALVE_TIME;
			i4Step														:= i4Step + 1;		
		END_IF
		
	9:
		
		bTimer1															:= TRUE;
	
		IF  r1.repres_valve_clear AND steam_iso_valve_clear THEN
			bTimer1														:= FALSE;
			rTime1														:= _STOPPING_TIME;
			i4Step														:= 98;
		ELSIF tonTimer1.Q THEN	
			bTimer1														:= FALSE;								
			sReactorError												:= SEL(r1.repres_valve_clear,gsRepressurizationValveError,'');
			sReactorError												:= SEL(steam_iso_valve_clear,gsSteamIsoValveError,sReactorError);

		END_IF
		
	
	80:																														// Manual process completing
		cycle_stage														:= 'repressurization.stopping';
		rTime1															:= _STOPPING_TIME;
		A_Reset();
		i4Step															:= 98;
		
	90:																														// Automatic process completing 
		cycle_stage														:= 'repressurization.stopping';
		rTime1															:= _STOPPING_TIME;
		A_Reset();
		i4Step															:= 98;
		
	98:
		bTimer1															:= TRUE;
		cycle_stage														:= 'repressurization.stopping';
		IF tonTimer1.Q THEN
			bTimer1														:= FALSE;
			i4Step														:= 99;
		END_IF
		
	99:
		bRepressurizationDone											:= TRUE;											// 5
		Current_Step													:= 0;
		i4Step															:= 0;
	
END_CASE

IF i4Step > 0 AND i4Step < 80 THEN
	iStep																:= i4Step;
	Current_Step														:= iStep;
	A_Check_Process();
	i4Step																:= iStep;
END_IF
END_ACTION

ACTION A4_Repressurization_1:
// Theseus - FB_Reactor_Set.A4_Repressurization_1
// Rev 1.0 - June 26, 2024

CASE i4Step OF
	
	0:	;
		
	1:
		cycle_stage														:= 'repressurization.initialize';
		rTime1															:= _VALVE_TIME;
		i4Step															:= i4Step + 1;
			
	2:
		cycle_stage														:= 'repressurization.running';
		bTimer1															:= TRUE;
		IF tonTimer1.Q THEN
			bTimer1														:= FALSE;
			i4Step														:= 98;
		END_IF
		
	80:																														// Manual process completing
		cycle_stage														:= 'repressurization.stopping.singlecycle';
		rTime1															:= _STOPPING_TIME;
		A_Reset();
		i4Step															:= 98;
		
	90:																														// Automatic process completing 
		cycle_stage														:= 'repressurization.stopping.multicycle';
		rTime1															:= _STOPPING_TIME;
		A_Reset();
		i4Step															:= 98;
		
	98:
		bTimer1															:= TRUE;
		//cycle_stage														:= 'repressurization.stopping';
		IF tonTimer1.Q THEN
			bTimer1														:= FALSE;
			i4Step														:= 99;
		END_IF
		

	99:
		bRepressurizationDone											:= TRUE;											// 5
		Current_Step													:= 0;
		i4Step															:= 0;
	
END_CASE

IF i4Step > 0 AND i4Step < 80 THEN
	iStep																:= i4Step;
	Current_Step														:= iStep;
	A_Check_Process();
	i4Step																:= iStep;
END_IF
END_ACTION

ACTION A4_Repressurization_OLD:
// Theseus - FB_Reactor_Set.A4_Repressurization
// Rev 1.0 - October 8, 2024

CASE i4Step OF
	
	0:	;
		
	1:
		cycle_stage														:= 'repressurization.initialize';
		sMessage														:= gsSystemCannotRun;
		IF P_U01.utility_error <> '' THEN
			sUtilityError												:= P_U01.utility_error;
		ELSIF r1.reactor_pres_error THEN
			sReactorError												:= gsReactorPresSensorError;
		ELSE
			A_Reset();																										// 1
			repres_valves												:= TRUE;											// 2		///@@@ Check clamps extended?
			steam_iso_valve												:= TRUE;
			rTime1														:= _VALVE_TIME;
			i4Step														:= i4Step + 1;
		END_IF
			
	2:
		bTimer1															:= TRUE;
		IF r1.repres_valve_clear AND steam_iso_valve_clear THEN
			bTimer1														:= FALSE;
			cycle_stage													:= 'repressurization.repressurize';
			rTime1														:= 5 * _MINUTES;
			i4Step														:= i4Step + 1;
		ELSIF tonTimer1.Q THEN
			sReactorError												:= SEL(r1.repres_valve_clear, gsRepressurizationValveError, gsSteamIsoValveError);
		END_IF

	3:
		bTimer1															:= TRUE;
		IF r1.reactor_pres > 0.98 AND r1.reactor_pres < 1.02 THEN															// 3
			bTimer1														:= FALSE;
			rTime1														:= 10 * _SECONDS;
			i4Step														:= i4Step + 1;
		ELSIF tonTimer1.Q THEN
			sReactorError												:= gsRepressurizationError;
		END_IF
		
	4:
		bTimer1															:= TRUE;
		IF tonTimer1.Q THEN																									// 4
			bTimer1														:= FALSE;
			i4Step														:= 99;
		END_IF
		
	
	80:																														// Manual process closing
		cycle_stage														:= 'repressurization.stopping';
		rTime1															:= _STOPPING_TIME;
		A_Reset();
		i4Step															:= 98;
		
	90:																														// Automatic process stopping
		cycle_stage														:= 'repressurization.stopping';
		rTime1															:= _STOPPING_TIME;
		A_Reset();
		i4Step															:= 98;
		
	98:
		bTimer1															:= TRUE;
		IF tonTimer1.Q THEN
			bTimer1														:= FALSE;
			i4Step														:= 99;
		END_IF
		
	99:
		bRepressurizationDone											:= TRUE;											// 5
		Current_Step													:= 0;
		i4Step															:= 0;
	
END_CASE

IF i4Step > 0 AND i4Step < 80 THEN
	iStep																:= i4Step;
	Current_Step														:= iStep;
	A_Check_Process();
	i4Step																:= iStep;
END_IF
END_ACTION

ACTION A5_Adsorption:
// Theseus - FB_Reactor_Set.A5_Adsorption
// Rev 1.0 - June 17, 2024

CASE i5Step OF	

	0:	;
		
	1:
		cycle_stage														:= 'adsorption.initialize';
		sMessage														:= gsSystemCannotRun;
		IF P_U01.utility_error <> '' THEN
			sUtilityError												:= P_U01.utility_error;
		ELSIF r1.reactor_pres_error THEN
			sReactorError												:= gsReactorPresSensorError;
		ELSE					
			retract_clamps												:= TRUE; 
			fan_setpoint												:= 0;
			steam_iso_valve												:= FALSE;      							// M01.XV07 <-TRUE
			P_U01.boiler_package 										:= FALSE;								// B01 : <- FALSE
			P_U01.steam_flow_control_valve_mode							:= eManual;
			P_U01.steam_flow_control_valve								:= _CLOSED;								// PCV02 <- CLOSE
			repres_valves												:= FALSE;								// R.XV02 <- TRUE
			dead_air_valve												:= FALSE;								// M01.XV04 <- FALSE
			steam_bypass_valve											:= FALSE;								// M01.XV08 <- FALSE
			product_iso_valve											:= FALSE;								// M01.XV05 <- FALSE
			P_U01.vacuum_pump_bypass_valve								:= TRUE;								// U01.XV04
			P_U01.product_line_ambient_valve							:= INT_TO_BOOL(eAmbient);				// U01.V11 <- ambient
			rTime1														:= 30 * _SECONDS;
			i5Step														:= i5Step + 1;												
		END_IF		
		
	2:
		
		bTimer1															:= TRUE;
		IF  inlet_clamps_retracted 					AND 
			outlet_clamps_retracted 				AND
			r1.fan_vfd_output = 0 					AND
			steam_iso_valve_clear					AND
			P_U01.steam_flow_control_valve_closed 	AND
			r1.repres_valve_clear					AND
			dead_air_valve_clear					AND
			steam_bypass_valve_clear				AND
			product_iso_valve_clear					AND
			P_U01.vacuum_pump_bypass_valve_clear 	AND
			P_U01.product_line_ambient_valve_clear 	AND 
			(r1.reactor_pres > 0.98 AND r1.reactor_pres < 1.02)  THEN
				
				bTimer1													:= FALSE; 
				rTime1													:= 5 * _SECONDS;
				i5Step													:= i5Step + 1; 
				
		ELSIF tonTimer1.Q THEN
			bTimer1														:= FALSE; 
			sReactorError												:= SEL(inlet_clamps_retracted,gsDoorClampsExtendedError,'');
			sReactorError												:= SEL(outlet_clamps_retracted,gsDoorClampsExtendedError,sReactorError);
			sReactorError												:= SEL(r1.fan_vfd_output <> 0,'fanVFDError',sReactorError);
			sReactorError												:= SEL(r1.repres_valve_clear,gsRepressurizationValveError,sReactorError);
			sReactorError												:= SEL(steam_iso_valve_clear,gsSteamIsoValveError,sReactorError);
			sReactorError												:= SEL(dead_air_valve_clear,gsDeadAirValveError,sReactorError);
			sReactorError												:= SEL(steam_bypass_valve_clear,gsSteamBypassValveError,sReactorError);
			sReactorError												:= SEL(product_iso_valve_clear,gsProductIsoValveError,sReactorError);
			sReactorError												:= SEL(r1.reactor_pres > 1.02, gsReactorPressureTooHighError ,sReactorError);
			sReactorError												:= SEL(r1.reactor_pres < 0.98, gsReactorPressureTooLowError ,sReactorError);
			
			sUtilityError												:= SEL(P_U01.vacuum_pump_bypass_valve_clear,'Vacuum Pump Bypass Valve Error ( U01.XV04)','');
			sUtilityError												:= SEL(P_U01.product_line_ambient_valve_clear,'Product Line Ambient Valve Error ( U01.XV11)',sUtilityError);
			sUtilityError												:= SEL(P_U01.steam_flow_control_valve_closed,gsSteamBypassValveError,sUtilityError);
		END_IF
		
	3: 
		bTimer1															:= TRUE;
		IF tonTimer1.Q THEN 
			bTimer1														:= FALSE;
			steam_iso_valve												:= TRUE;      							// M01.XV07 <-TRUE
			repres_valves												:= TRUE;								// R.XV02 <- TRUE
			rTime1														:= _VALVE_TIME;
			i5Step														:= i5Step + 1; 
		END_IF
		
	4: 
		bTimer1															:= TRUE;
		IF steam_iso_valve_clear AND r1.repres_valve_clear THEN
			bTimer1														:= FALSE;
			open_doors													:= TRUE;
			rTime1														:= _DOOR_ACTUATION_TIMEOUT;
			i5Step														:= i5Step + 1; 
		ELSIF tonTimer1.Q THEN
			bTimer1														:= FALSE;
			sReactorError												:= SEL(dead_air_valve_clear,gsDeadAirValveError,'');
			sReactorError												:= SEL(r1.repres_valve_clear,gsRepressurizationValveError,sReactorError);
		END_IF
		
		
	5: 
		
		bTimer1															:= TRUE;
			
		IF inlet_doors_open AND outlet_doors_open THEN	
			bTimer1														:= FALSE; 		
			fan_setpoint												:= P_M01.SP_reactor_set_1_vfd_percent;
			steam_iso_valve												:= FALSE; 
			repres_valves												:= FALSE;
			rTime1														:= _FAN_RS_DELAY_TIME;
			i5Step														:= i5Step + 1; 
		ELSIF tonTimer1.Q THEN
			bTimer1														:= FALSE; 
			sReactorError												:= gsDoorsNotOpenError;
		END_IF 
	
	6: 
		cycle_stage														:= 'adsorption.adsorption_started';
		bTimer1															:= TRUE;
		rTime2															:= P_M01.SP_adsorption_duration * _MINUTES;
		bTimer2															:= TRUE;
		bPass1															:= r1.fan_vfd_output >= fan_setpoint * 0.9 AND r1.fan_vfd_output <= fan_setpoint * 1.1;
		IF 	steam_iso_valve_clear AND
			r1.repres_valve_clear AND
			(r1.fan_vfd_output >= fan_setpoint * 0.9 AND r1.fan_vfd_output <= fan_setpoint * 1.1) THEN
			
				bTimer1													:= FALSE; 
				rTime1													:= 120 * _SECONDS;
				i5Step													:= i5Step + 1; 
				
		ELSIF tonTimer1.Q THEN
			bTimer1														:= FALSE; 
			sReactorError												:= SEL(bPass1,'Fan did not reach the set speed +/- 10%','');
			sReactorError												:= SEL(steam_iso_valve_clear,gsSteamControlValveError,sReactorError);
			sReactorError												:= SEL(r1.repres_valve_clear,gsRepressurizationValveError ,sReactorError);
		END_IF

	7: 
		
		bTimer1															:= TRUE;
		IF sorbent_average_temp < 40 THEN
			bTimer1														:= FALSE; 
			reactor_drain_adsorption_on									:= TRUE;
			rTime1														:= 120 * _SECONDS;
			i5Step														:= i5Step + 1; 
		ELSIF tonTimer1.Q THEN
			sReactorError												:= 'Evac Sorbent did not cool down enough at beginning of desorption';		
		END_IF
		
	8:   // new step
		
		IF NOT reactor_drain_adsorption_on THEN
			bTimer1														:= TRUE;
		END_IF
		IF tonTimer1.Q THEN
			bTimer1														:= FALSE;
			P_U01.condenser_knockout_drain_adsorption_on				:= TRUE;
			i5Step														:= i5Step + 1; 
		END_IF
		IF tonTimer2.Q THEN
			i5Step														:= i5Step + 1; 
		END_IF
		
	9: 
		
		IF tonTimer2.Q THEN
			bTimer2														:= FALSE; 
			fan_setpoint												:= 0;
			rTime1														:= 30 * _SECONDS;
			i5Step														:= i5Step + 1; 
		END_IF
		
	10: 
		
		
		bTimer1															:= TRUE;
		IF r1.fan_vfd_output = 0 AND tonTimer1.Q THEN
			bTimer1														:= FALSE; 
			close_doors													:= TRUE;
			rTime1														:= _DOOR_ACTUATION_TIMEOUT;
			i5Step														:= i5Step + 1; 
		ELSIF r1.fan_vfd_output <> 0 AND tonTimer1.Q THEN
			bTimer1														:= FALSE; 
			sReactorError												:= 'Adsorption Fan VFD did not turn off';	
		END_IF
		
	11:
		cycle_stage														:= 'adsorption.stopping ';
		
		bTimer1															:= TRUE;
		
		IF inlet_doors_closed AND outlet_doors_closed THEN
			bTimer1														:= FALSE; 
			P_U01.vacuum_pump_bypass_valve								:= FALSE;								// U01.XV04
			rTime1														:= _VALVE_TIME;
			i5Step														:= i5Step + 1; 
		
		ELSIF tonTimer1.Q THEN
			bTimer1														:= FALSE; 
			sReactorError												:= gsDoorsNotClosedError;
		END_IF
		
	12:
		
		bTimer1															:= TRUE;
				
		IF P_U01.vacuum_pump_bypass_valve_clear THEN
			bTimer1														:= FALSE; 
			rTime1														:= _STOPPING_TIME;
			i5Step														:= 98;
		ELSIF tonTimer1.Q THEN	
			bTimer1														:= FALSE; 	
			sReactorError												:= 'Vacuum Pump Bypass Error ( U01.XV04)';
		END_IF
		
	80:																														// Manual process completing
		cycle_stage														:= 'adsorption.stopping';
		rTime1															:= _STOPPING_TIME;
		A_Reset();
		i5Step															:= 98;
		
	90:																														// Automatic process completing 
		cycle_stage														:= 'adsorption.stopping';
		rTime1															:= _STOPPING_TIME;
		A_Reset();
		i5Step															:= 98;
		
	98:
		cycle_stage														:= 'adsorption.stopping';
		bTimer1															:= TRUE;
		IF tonTimer1.Q THEN
			bTimer1														:= FALSE;
			i5Step														:= 99;
		END_IF
		
	99:
		bAdsorptionDone													:= TRUE;											
		Current_Step													:= 0;
		i5Step															:= 0;	
	
END_CASE

IF i5Step > 0 AND i5Step < 80 THEN
	iStep																:= i5Step;
	Current_Step														:= iStep;
	A_Check_Process();
	i5Step																:= iStep;
END_IF
END_ACTION

ACTION A5_Adsorption_1:
// Theseus - FB_Reactor_Set.A5_Adsorption_1
// Rev 1.0 - June 26, 2024

CASE i5Step OF	

	0:	;
		
	1:
		cycle_stage														:= 'adsorption.initialize';
		rTime1															:= _VALVE_TIME;
		i5Step															:= i5Step + 1;
		
	2:
		cycle_stage														:= 'adsorption.initialize';
		bTimer1															:= TRUE;
		IF tonTimer1.Q THEN
			bTimer1														:= FALSE;
			i5Step														:= 98;
		END_IF
		
		
	80:																														// Manual process completing
		cycle_stage														:= 'adsorption.stopping';
		rTime1															:= _STOPPING_TIME;
		A_Reset();
		i5Step															:= 98;
		
	90:																														// Automatic process completing 
		cycle_stage														:= 'adsorption.stopping';
		rTime1															:= _STOPPING_TIME;
		A_Reset();
		i5Step															:= 98;
		
	98:
		cycle_stage														:= 'adsorption.stopping';
		bTimer1															:= TRUE;
		IF tonTimer1.Q THEN
			bTimer1														:= FALSE;
			i5Step														:= 99;
		END_IF
		
	
	99:
		cycle_stage														:= 'adsorption.completed';
		bAdsorptionDone													:= TRUE;											
		Current_Step													:= 0;
		i5Step															:= 0;
	
END_CASE

IF i5Step > 0 AND i5Step < 80 THEN
	iStep																:= i5Step;
	Current_Step														:= iStep;
	A_Check_Process();
	i5Step																:= iStep;
END_IF
END_ACTION

ACTION A5_Adsorption_OLD:
// Theseus - FB_Reactor_Set.A5_Adsorption
// Rev 1.0 - June 17, 2024

CASE i5Step OF	

	0:	;
		
	1:
		i5Step															:= 0;
	
END_CASE

IF i5Step > 0 AND i5Step < 80 THEN
	iStep																:= i5Step;
	Current_Step														:= iStep;
	A_Check_Process();
	i5Step																:= iStep;
END_IF
END_ACTION

ACTION A6_Evacuation:
// Theseus - FB_Reactor_Set.A6_Evacuation
// Rev 1.0 - December 3, 2024

CASE i6Step OF
	
	0:	;
	
	1:
		cycle_stage														:= 'evacuation.initialize';
		sMessage														:= gsSystemCannotRun;
		//gbGasketsActivated											:= FALSE;
		IF sorbent_high_temp < 60 THEN
			i6Step															:= i6Step + 1;										
		ELSE
			sReactorError												:= 'Sorbent too hot for dead air evacuation';
		END_IF
		
		
	2:
		//A_Reset();																											
		steam_bypass_valve												:= FALSE;								// M01.XV08 <- FALSE
		steam_iso_valve													:= FALSE;      							// M01.XV07 <-TRUE
		product_iso_valve												:= FALSE;								// M01.XV05 <- FALSE
		fan_setpoint													:= 0;
		P_U01.vacuum_pres_control_valve_mode							:= eManual;
		P_U01.vacuum_pres_control_valve									:= _CLOSED;
		P_U01.steam_flow_control_valve_mode								:= eManual;
		P_U01.steam_flow_control_valve									:= _CLOSED;
		P_U01.product_line_ambient_valve								:= FALSE;
		P_U01.vacuum_pump_bypass_valve									:= FALSE;								// U01.XV04
		P_U01.vacuum_pump_inlet_valve									:= FALSE;
//		P_U01.drainage_on												:= TRUE;
		rTime1															:= _VALVE_TIME;
		i6Step															:= i6Step + 1;
		
	3:
		bTimer1															:= TRUE;
		bPass1															:= steam_bypass_valve_clear;
		bPass2															:= steam_iso_valve_clear;
		bPass3															:= product_iso_valve_clear;
		bPass4															:= r1.fan_vfd_output = 0;
		bPass5															:= P_U01.vacuum_pres_control_valve_closed;
		bPass6															:= P_U01.steam_flow_control_valve_closed;
		bPass7															:= P_U01.product_line_ambient_valve_clear;
		bPass8															:= P_U01.vacuum_pump_bypass_valve_clear;
		bPass9															:= P_U01.vacuum_pump_inlet_valve_clear;
		IF bPass1 AND bPass2 AND bPass3 AND bPass4 AND bPass5 AND bPass6 AND bPass7 AND bPass8 AND bPass9 THEN
			bTimer1														:= FALSE;
			rTime1														:= _SECONDS * 60;
			i6Step														:= i6Step + 1;
		ELSIF tonTimer1.Q THEN
			bTimer1														:= FALSE;
			sReactorError												:= SEL(bPass1,'Steam Bypass Valve Error RS XV08', '');
			sReactorError												:= SEL(bPass2, gsSteamIsoValveError, sReactorError);
			sReactorError												:= SEL(bPass3, gsProductIsoValveError, sReactorError);
			sReactorError												:= SEL(bPass4, 'Fan VFD SP Error', sReactorError);
			sUtilityError												:= SEL(bPass5, gsVacuumPressureControlValveError, '');
			sUtilityError												:= SEL(bPass6, gsSteamFlowConrolValveError, sUtilityError);
			sUtilityError												:= SEL(bPass7, gsProductLineAmbientValveError, sUtilityError);
			sUtilityError												:= SEL(bPass8, gsVacuumPumpBypassValveError, sUtilityError);
			sUtilityError												:= SEL(bPass9, gsVacuumPumpInletValveError, sUtilityError);
		END_IF
		
	4:
		bTimer1															:= TRUE;
		bPass1															:= r1.reactor_pres > P_M01.SP_evacuation_ideal_pressure;
		bPass2															:= NOT reactor_drain_vessel_lsh;
		bPass3															:= NOT P_U01.product_condensate_drum_lsh;
//		bPass4															:= P_U01.vacuum_separator_level > P_U01.SP_vacuum_separator_level_low;
		IF bPass1 AND bPass2 AND bPass3  THEN
			bTimer1														:= FALSE;
			cycle_stage													:= 'evacuation.starting';
			P_U01.drainage_on											:= FALSE;											
			i6Step														:= i6Step + 1;
		ELSIF tonTimer1.Q THEN
			bTimer1														:= FALSE;
			sReactorError												:= SEL(bPass1, gsReactorPressureTooLowError, '');
			sReactorError												:= SEL(bPass2, gsReactorDrainError, sReactorError);
			sUtilityError												:= SEL(bPass3, gsProductCondensateDrumLshError, '');
		END_IF
	
	5:
		
			rTime1														:= _CLAMP_ACTUATION_TIMEOUT;
			P_U01.vacuum_liquid_pump									:= TRUE;											
			P_U01.vacuum_liquid_loop_fan								:= TRUE;
			retract_clamps												:= TRUE;											
			i6Step														:= i6Step + 1;
		
	6:
		bTimer1															:= TRUE;
		IF inlet_clamps_retracted AND outlet_clamps_retracted THEN
			bTimer1														:= FALSE;
			close_doors													:= TRUE;											
			rTime1														:= _DOOR_ACTUATION_TIMEOUT;
			i6Step														:= i6Step + 1;
		ELSIF tonTimer1.Q THEN
			bTimer1														:= FALSE;
			sReactorError												:= SEL(inlet_clamps_retracted, gsInletDoorClampsRetractedError, '');
			sReactorError												:= SEL(outlet_clamps_retracted, gsOutletDoorClampsRetractedError, sReactorError);
		END_IF

	7:
		bTimer1															:= TRUE;
		IF inlet_doors_closed AND outlet_doors_closed THEN
			bTimer1														:= FALSE;
			extend_clamps												:= TRUE;											
			rTime1														:= 30 * _SECONDS;
			i6Step														:= i6Step + 1;
		ELSIF tonTimer1.Q THEN
			sReactorError												:= gsDoorsNotClosedError;
			bTimer1														:= FALSE;
		END_IF

	8:
		cycle_stage														:= 'evacuation.vacuum_init';
		bTimer1															:= TRUE;
		bPass1															:= P_U01.vacuum_pump_water_flow > P_U01.SP_minimum_vacuum_cooling_loop_flow;
		bPass2															:= P_U01.vacuum_pump_water_temp_1 < P_U01.SP_max_vacuum_cooling_loop_temp;
		IF bPass1 AND bPass2 THEN																							
			bTimer1														:= FALSE;
			cycle_stage													:= 'evacuation.evacuation';
			P_U01.dead_air_inlet_valve									:= TRUE;
			P_U01.vacuum_pump											:= TRUE;
			rTime1														:= 20 * _SECONDS;
			i6Step														:= i6Step + 1;
		ELSIF tonTimer1.Q THEN
			bTimer1														:= FALSE;
			sUtilityError												:= SEL(bPass1, gsVacuumCoolingLoopFlowError, '');
			sUtilityError												:= SEL(bPass2, gsVacuumCoolingLoopTempError, sUtilityError);
		END_IF
			
	9:
		bTimer1															:= TRUE;
		bPass1															:= P_U01.product_vacuum_pres <= P_U01.SP_minimum_dead_air_line_pressure;
		IF P_U01.dead_air_inlet_valve_clear AND bPass1 THEN
			bTimer1														:= FALSE;						
			dead_air_valve												:= TRUE;
			rTime1														:= _VALVE_TIME;
			i6Step														:= i6Step + 1;
		ELSIF tonTimer1.Q THEN
			bTimer1														:= FALSE;
			sUtilityError												:= SEL(P_U01.dead_air_inlet_valve_clear,gsDeadAirInletValveError,'');
			sUtilityError												:= SEL(bPass1,gsDeadAirLinePressureError,sUtilityError);
		END_IF
	
	10:
		bTimer1															:= TRUE;	
		IF dead_air_valve_clear	THEN
			bTimer1														:= FALSE;
			rTime1														:= P_M01.SP_evacuation_duration * _MINUTES;
			i6Step														:= i6Step + 1;
		ELSIF tonTimer1.Q THEN
			sReactorError												:= gsDeadAirValveError;
			bTimer1														:= FALSE;
		END_IF
	
	11:
		bTimer1															:= TRUE;
		IF r1.reactor_pres <= P_M01.SP_evacuation_ideal_pressure  THEN														
			bTimer1														:= FALSE;
//			rReactorLeakTestStartingPressure							:= r1.reactor_pres;
			dead_air_valve												:= FALSE;
			P_U01.dead_air_inlet_valve									:= FALSE;
			P_U01.vacuum_pump											:= FALSE;
			P_U01.vacuum_liquid_pump									:= FALSE;
			P_U01.vacuum_liquid_loop_fan								:= FALSE;
			rTime1														:= _VALVE_TIME;
			i6Step														:= i6Step + 1;
		ELSIF tonTimer1.Q THEN
			bTimer1														:= FALSE;
			sReactorError												:= gsReactorPressureTooHighError;
		END_IF
		
	12:
		bTimer1															:= TRUE;
		IF dead_air_valve_clear AND P_U01.dead_air_inlet_valve_clear  AND inlet_clamps_extended AND outlet_clamps_extended THEN																						// 10
			bTimer1														:= FALSE;
			rTime1														:= P_M01.SP_vacuum_leak_test_duration * _MINUTES;
			i6Step														:= i6Step + 1;
		ELSIF tonTimer1.Q THEN
			bTimer1														:= FALSE;
			sReactorError												:= SEL(dead_air_valve_clear,gsDeadAirValveError,'');
			sUtilityError												:= gsDeadAirInletValveError;
			sReactorError												:= SEL(inlet_clamps_extended, gsInletDoorClampsExtendedError, '');
			sReactorError												:= SEL(outlet_clamps_extended, gsOutletDoorClampsExtendedError, sReactorError);
		END_IF
		
	13: //mm
		bTimer1															:= TRUE;
		IF tonTimer1.Q THEN
//			reactor_test_leakage_pressure									:= r1.reactor_pres - rReactorLeakTestStartingPressure;
			IF r1.reactor_pres  <= P_M01.SP_evacuation_ideal_pressure * 1.1 THEN									// 11
				bTimer1													:= FALSE;
				rTime1													:= _STOPPING_TIME;
				i6Step													:= 98;
			ELSE
				bTimer1													:= FALSE;
				sReactorError											:= gsUnacceptableReactorLeakRate;
			END_IF
		END_IF
		
	

	80:																														// Stop process individually 
		cycle_stage														:= 'evacuation.stopping';
		dead_air_valve													:= FALSE;											
		P_U01.dead_air_inlet_valve										:= FALSE;
		P_U01.vacuum_pump												:= FALSE;
		P_U01.vacuum_liquid_pump										:= FALSE;
		P_U01.vacuum_liquid_loop_fan									:= FALSE;
		A_Reset();
		rTime1															:= _STOPPING_TIME;
		i6Step															:= 98;
		
	90:																														// Automatic process stopping
		cycle_stage														:= 'evacuation.stopping';
		A_Reset();
		rTime1															:= _STOPPING_TIME;
		i6Step															:= 98;
		
	98:
		cycle_stage														:= 'evacuation.stopping';
		bTimer1															:= TRUE;
		IF tonTimer1.Q THEN
			bTimer1														:= FALSE;
			i6Step														:= 99;
		END_IF
		
	99:
		bEvacuationDone													:= TRUE;											// 13
		Current_Step													:= 0;
		i6Step															:= 0;
	
END_CASE

IF i6Step > 0 AND i6Step < 80 THEN
	iStep																:= i6Step;
	Current_Step														:= iStep;
	sReactorError														:= SEL(r1.reactor_pres_error, sReactorError, gsReactorPresSensorError);
	sUtilityError														:= SEL(P_U01.vacuum_separator_level_error, sUtilityError, gsVacuumSeparatorLevelSensorError);
	sUtilityError														:= SEL(P_U01.vacuum_pump_water_flow_error, sUtilityError, gsVacuumPumpWaterFlowSensorError);
	sUtilityError														:= SEL(P_U01.vacuum_pump_water_temp_1_error, sUtilityError, gsVacuumPumpWaterTemp1SensorError);
	A_Check_Process();
	i6Step																:= iStep;
END_IF
END_ACTION

ACTION A6_Evacuation_1:

CASE i6Step OF	

	0:	;
		
	1:
		cycle_stage														:= 'evacuation.initialize';
		rTime1															:= _VALVE_TIME;
		i6Step															:= i6Step + 1;
		
	2:
		cycle_stage														:= 'evacuation.started';
		bTimer1															:= TRUE;
		IF tonTimer1.Q THEN
			bTimer1														:= FALSE;
			i6Step														:= 98;
		END_IF
		
	80:																														// Stop process individually 
		cycle_stage														:= 'evacuation.stopping';
		rTime1															:= _STOPPING_TIME;
		i6Step															:= 98;
		
	90:																														// Automatic process stopping
		cycle_stage														:= 'evacuation.stopping';
		rTime1															:= _STOPPING_TIME;
		i6Step															:= 98;
		
	98:
		cycle_stage														:= 'evacuation.stopping';
		bTimer1															:= TRUE;
		IF tonTimer1.Q THEN
			bTimer1														:= FALSE;
			i6Step														:= 99;
		END_IF
	99:
		cycle_stage														:= 'evacuation.completed';
		bEvacuationDone													:= TRUE;											// 5
		Current_Step													:= 0;
		i6Step															:= 0;
	
END_CASE

IF i6Step > 0 AND i6Step < 80 THEN
	iStep																:= i6Step;
	Current_Step														:= iStep;
	A_Check_Process();
	i6Step																:= iStep;
END_IF
END_ACTION

ACTION A6_Evacuation_OLD:
// Theseus - FB_Reactor_Set.A6_Evacuation
// Rev 1.0 - October 9, 2024

CASE i6Step OF
	
	0:	;
	
	1:
		cycle_stage														:= 'evacuation.initialize';
		giEvacuationCounter												:= giEvacuationCounter - 1;
		sMessage														:= gsSystemCannotRun;
		gbGasketsActivated												:= FALSE;
		IF P_U01.utility_error <> '' THEN
			sUtilityError												:= P_U01.utility_error;
		ELSIF product_line_pres_error THEN
			sReactorError												:= gsProductLinePressureSensorError;
		ELSIF r1.reactor_pres_error THEN
			sReactorError												:= gsReactorPresSensorError;
		ELSIF inlet_clamps_extended AND outlet_clamps_extended THEN
			i6Step														:= i6Step + 3;
			rTime1														:= 1 * _SECONDS;
		ELSE
			A_Reset();																										// 1
			retract_clamps												:= TRUE;											// 2
			rTime1														:= _CLAMP_ACTUATION_TIMEOUT; 		// Use Valve time if longer
			i6Step														:= i6Step + 1;
		END_IF
		
	2:
		bTimer1															:= TRUE;
		cycle_stage														:= 'evacuation.close_valve_doors';
		IF rs_valves_clear AND inlet_clamps_extended AND outlet_clamps_extended THEN
			bTimer1														:= FALSE;
			close_doors													:= TRUE;
			rTime1														:= _DOOR_ACTUATION_TIMEOUT;
			i6Step														:= i6Step + 1;
		ELSIF tonTimer1.Q THEN
			IF inlet_clamps_extended AND outlet_clamps_extended THEN
				sReactorError											:= SEL(dead_air_valve_clear, gsDeadAirValveError, '');
				sReactorError											:= SEL(product_iso_valve_clear, gsProductIsoValveError, sReactorError);
				sReactorError											:= SEL(condensate_valve_clear, gsCondensateValveError, sReactorError);
				sReactorError											:= SEL(steam_iso_valve_clear, gsSteamIsoValveError, sReactorError);
				sReactorError											:= SEL(steam_bypass_valve_clear, gsSteamBypassValveError, sReactorError);
			ELSE
				sReactorError											:= SEL(NOT inlet_clamps_extended, '', gsInletDoorClampsExtendedError);
				sReactorError											:= SEL(outlet_clamps_extended, sReactorError, gsOutletDoorClampsExtendedError);
			END_IF
		END_IF

	3:
		bTimer1															:= TRUE;
		IF (inlet_doors_closed AND outlet_doors_closed) OR r1.reactor_pres < 0.9 THEN				// smrg debug - allow test to continue if picking up where previous vacuum test left off (doors may not show up as closed under vacuum)
			bTimer1														:= FALSE;
			extend_clamps												:= TRUE;
			rTime1														:= _CLAMP_ACTUATION_TIMEOUT;
			i6Step														:= i6Step + 1;
		ELSIF tonTimer1.Q THEN
			sReactorError												:= gsDoorsNotClosedError;
		END_IF

	4:
		bTimer1															:= TRUE;
		IF tonTimer1.Q THEN
			bTimer1														:= FALSE;
			P_U01.dead_air_inlet_valve									:= TRUE;											// 5
			P_U01.product_line_ambient_valve							:= INT_TO_BOOL(eAmbient);	
			P_U01.vacuum_liquid_loop_fan								:= TRUE;
			P_U01.vacuum_liquid_pump									:= TRUE;
			repres_valves												:= FALSE;
			steam_iso_valve												:= FALSE;
			rTime1														:= 5 * _SECONDS;									// give water time to start flowing before attempting to turn on vacuum pump
			i6Step														:= i6Step + 1;
		END_IF
		
	5:
		bTimer1															:= TRUE;
		IF tonTimer1.Q THEN
			bTimer1														:= FALSE;
			rTime1														:= _VALVE_TIME;
			i6Step														:= i6Step + 1;
		END_IF
		
	6:		
		cycle_stage														:= 'evacuation.vacuum_init';
		bTimer1															:= TRUE;
		//IF P_U01.dead_air_inlet_valve_clear AND P_U01.product_line_ambient_valve_clear THEN
		IF P_U01.dead_air_inlet_valve_clear THEN								// smrg debug
			bTimer1														:= FALSE;
			P_U01.vacuum_pump											:= TRUE;											// 6
			cycle_stage													:= 'evacuation.evacuation';
			rTime1														:= 60 * _SECONDS;
			i6Step														:= i6Step + 1;
		ELSIF tonTimer1.Q THEN
			sReactorError												:= SEL(dead_air_valve_clear, gsDeadAirValveError, '');
			sReactorError												:= SEL(P_U01.product_line_ambient_valve_clear, gsProductLineAmbientValveError, sReactorError);
		END_IF
		
	7:
		bTimer1															:= TRUE;
		IF P_U01.product_vacuum_pres <= P_M01.SP_evacuation_ideal_pressure THEN													// 7
			bTimer1														:= FALSE;
			dead_air_valve												:= TRUE;											// 8		
			rTime1														:= _VALVE_TIME;
			i6Step														:= i6Step + 1;
		ELSIF tonTimer1.Q THEN
			sReactorError												:= gsDeadAirValveError;
		END_IF
		
	8:
		bTimer1															:= TRUE;
		IF dead_air_valve_clear THEN													
			rTime1														:= P_M01.SP_evacuation_duration * _MINUTES;
			bTimer1														:= FALSE;										
			i6Step														:= i6Step + 1;
		ELSIF tonTimer1.Q THEN
			sReactorError												:= gsVacuumLinePressureHighError;
		END_IF
	
	9:
		bTimer1															:= TRUE;
		IF r1.reactor_pres <= P_M01.SP_evacuation_ideal_pressure THEN														// 9
			bTimer1														:= FALSE;
			i6Step														:= i6Step + 1;
		ELSIF tonTimer1.Q THEN
			sReactorError												:= gsReactorPressureTooHighError;
		END_IF

	10:
		IF inlet_clamps_extended AND outlet_clamps_extended THEN																						
			gbGasketsActivated											:= TRUE;											// 10
			dead_air_valve												:= FALSE;											// 11
			P_U01.vacuum_liquid_loop_fan								:= FALSE;
			P_U01.vacuum_liquid_pump									:= FALSE;
			P_U01.vacuum_pump											:= FALSE;
			rTime1														:= _VALVE_TIME;
			i6Step														:= i6Step + 1;
		ELSE
			sReactorError												:= SEL(NOT inlet_clamps_extended, '', gsInletDoorClampsExtendedError);
			sReactorError												:= SEL(NOT outlet_clamps_extended, sReactorError, gsOutletDoorClampsExtendedError);
		END_IF		
		
	11:
		bTimer1															:= TRUE;
		IF dead_air_valve_clear THEN
			bTimer1														:= FALSE;
			IF gbFirstEvacuation THEN																						// 12
				gbFirstEvacuation										:= FALSE;
				cycle_stage												:= 'evacuation.settle_time';
				rTime1													:= P_M01.SP_vacuum_settle_time * _MINUTES;			// 13
				i6Step													:= i6Step + 1;
			ELSE																											// if not first evacuation, skip leak check
				i6Step													:= 13;
			END_IF
		ELSIF tonTimer1.Q THEN
			sReactorError												:= gsDeadAirValveError;
		END_IF

	12:
		bTimer1															:= TRUE;
		IF tonTimer1.Q THEN	
			bTimer1														:= FALSE;			
			cycle_stage													:= 'evacuation.leak_check';
			rR1SavedPressure											:= r1.reactor_pres;									// 14
			rTime1														:= P_M01.SP_vacuum_leak_test_duration * _MINUTES;
			i6Step														:= i6Step + 1;
		END_IF
		
	13:
		bTimer1															:= TRUE;
		IF tonTimer1.Q THEN																									// 15
			bTimer1														:= FALSE;
			rR1Leakage													:= (r1.reactor_pres - rR1SavedPressure) / P_M01.SP_vacuum_leak_test_duration;
			IF rR1Leakage < P_M01.SP_unacceptable_vacuum_pressure_change THEN												// 16
				bVacuumHolding											:= TRUE;
				i6Step													:= i6Step + 1;
			ELSE
				bVacuumHolding											:= FALSE;
				sReactorError											:= gsVacuumPressureUnacceptableError;
			END_IF
		END_IF

	14:
		IF (giEvacuationCounter = 0) THEN																					// 17
			retract_clamps												:= TRUE;											// 18
			rTime1														:= _CLAMP_ACTUATION_TIMEOUT;
			i6Step														:= i6Step + 1;
		ELSE
			i6Step														:= 99;
		END_IF
 
	15:
		bTimer1															:= TRUE;
		IF inlet_clamps_retracted AND outlet_clamps_retracted THEN
			i6Step														:= 99;
		ELSIF tonTimer1.Q THEN
			sReactorError												:= gsDoorClampsExtendedError;
			sMessage													:= gsSystemWillStop;
		END_IF
		
	80:																														// Stop process
		cycle_stage														:= 'evacuation.stopping';
		A_Reset();
		rTime1															:= _STOPPING_TIME;
		i6Step															:= 98;
		
	90:																														// Automatic process stopping
		cycle_stage														:= 'evacuation.stopping';
		A_Reset();
		rTime1															:= _STOPPING_TIME;
		i6Step															:= 98;
		
	98:
		bTimer1															:= TRUE;
		IF tonTimer1.Q THEN
			bTimer1														:= FALSE;
			i6Step														:= 99;
		END_IF
		
	99:
		bEvacuationDone													:= TRUE;											// 19
		Current_Step													:= 0;
		i6Step															:= 0;
	
END_CASE

IF i6Step > 0 AND i6Step < 80 THEN
	iStep																:= i6Step;
	Current_Step														:= iStep;
	A_Check_Process();
	i6Step																:= iStep;
END_IF
END_ACTION

ACTION A7_Desorption:
// Theseus - FB_Reactor_Set.A7_Desorption_1
// Rev 1.0 - June 24, 2024

CASE i7Step OF
	
	0:	;
		
	1:
		
		cycle_stage														:= 'desorption.initialize';
		sMessage														:= gsSystemCannotRun;
		
		IF P_U01.utility_error <> '' THEN
			sUtilityError												:= P_U01.utility_error;
		ELSIF r1.reactor_pres_error THEN
			sReactorError												:= gsReactorPresSensorError;
		ELSE			
			A_Reset();
			P_U01.boiler_package 										:= FALSE;
//			P_U01.vacuum_pres_control_valve								:= _CLOSED;											//add it as input to P_U01			
			rTime1															:= _VALVE_TIME;
			i7Step															:= i7Step + 1;										
		END_IF		
		
		
	2:
		rTime1															:= _VALVE_TIME;
		bTimer1															:= TRUE;
		IF rs_valves_clear AND P_U01.vacuum_pres_control_valve_closed  THEN
			bTimer1														:= FALSE; 
			i7Step														:= i7Step + 1;
		ELSIF tonTimer1.Q THEN
			sReactorError												:= gsProcessCannotContinue;
		END_IF	
	
	3: //excel sheet step2 - open repres valve
		cycle_stage														:= 'desorption.running';
		r1.repres_valve													:= TRUE;
		rTime1															:= _VALVE_TIME;
		bTimer1															:= TRUE;
		IF R1.repres_valve_clear THEN
			bTimer1														:= FALSE;
			i7Step														:= i7Step + 1;
		ELSIF tonTimer1.Q THEN
			sReactorError												:= gsRepressurizationValveError;
		END_IF

	4: //excel sheet step 3 - wait for repressurization
		rTime1															:= 5 * _MINUTES;
		bTimer1															:= TRUE;
		IF r1.reactor_pres > 0.98 AND r1.reactor_pres < 1.02 THEN
			bTimer1														:= FALSE;
			i7Step														:= i7Step + 1;
		ELSIF tonTimer1.Q THEN
			sReactorError												:= gsRepressurizationError;
		END_IF
		
	5: //excel sheet step 4 - settle time
		rTime2															:=10 * _SECONDS;
		bTimer2															:= TRUE;
		IF tonTimer2.Q THEN
			bTimer2														:= FALSE;
			i7Step														:= 99;
		END_IF
		
	80:																														// Manual process completing
		cycle_stage														:= 'desorption.stopping';
		rTime1															:= _STOPPING_TIME;
		A_Reset();
		i7Step															:= 98;
		
	90:																														// Automatic process completing 
		cycle_stage														:= 'desorption.stopping';
		rTime1															:= _STOPPING_TIME;
		A_Reset();
		i7Step															:= 98;
		
	98:
		bTimer1															:= TRUE;
		IF tonTimer1.Q THEN
			bTimer1														:= FALSE;
			i7Step														:= 99;
		END_IF
			
		
	99:
		bDesorptionDone													:= TRUE;											// 19
		Current_Step													:= 0;
		i7Step															:= 0;
	
END_CASE

IF i7Step > 0 AND i7Step < 80 THEN
	iStep																:= i7Step;
	Current_Step														:= iStep;
	A_Check_Process();
	i7Step																:= iStep;
END_IF
END_ACTION

ACTION A7_Desorption_1:
// Theseus - FB_Reactor_Set.A7_Desorption_1
// Rev 1.0 - June 24, 2024

CASE i7Step OF
	
	0:	;
		
	1:
		rTime1															:= _VALVE_TIME;
		i7Step															:= i7Step + 1;
		
	2:
		bTimer1															:= TRUE;
		IF tonTimer1.Q THEN
			bTimer1														:= FALSE;
			i7Step														:= 99;
		END_IF

	99:
		bDesorptionDone													:= TRUE;											// 19
		Current_Step													:= 0;
		i7Step															:= 0;
	
END_CASE

IF i7Step > 0 AND i7Step < 80 THEN
	iStep																:= i7Step;
	Current_Step														:= iStep;
	A_Check_Process();
	i7Step																:= iStep;
END_IF
END_ACTION

ACTION A7_Desorption_OLD:
// Theseus - FB_Reactor_Set.A7_Desorption
// Rev 1.0 - June 17, 2024

CASE i7Step OF
	
	0:	;
		
	1:
		i7Step															:= 0;
	
END_CASE

IF i7Step > 0 AND i7Step < 80 THEN
	iStep																:= i7Step;
	Current_Step														:= iStep;
	A_Check_Process();
	i7Step																:= iStep;
END_IF
END_ACTION

ACTION A8_Bypass:
// Theseus - FB_Reactor_Set.A8_Bypass
// Rev 1.0 - December 3, 2024

CASE i8Step OF
	
	0:	;
	
	1:
		cycle_stage														:= 'bypass.initialize';
		sMessage														:= gsSystemCannotRun;
		i8Step															:= i8Step + 1;										// Run first step to check for sensor errors
		
	2:
		A_Reset();																											// 1
		P_U01.vacuum_pres_control_valve_mode							:= eManual;
		P_U01.vacuum_pres_control_valve									:= _CLOSED;
		P_U01.steam_flow_control_valve_mode								:= eManual;
		P_U01.steam_flow_control_valve									:= _CLOSED;
		P_U01.product_line_ambient_valve								:= FALSE;
		P_U01.vacuum_pump_inlet_valve									:= FALSE;
		P_U01.vacuum_pump_bypass_valve									:= TRUE;
		P_U01.drainage_on												:= TRUE;
		rTime1															:= _VALVE_TIME;
		i8Step															:= i8Step + 1;
		
	3:
		bTimer1															:= TRUE;
		bPass1															:= P_U01.vacuum_pres_control_valve_closed;
		bPass2															:= P_U01.steam_flow_control_valve_closed;
		bPass3															:= P_U01.product_line_ambient_valve_clear;
		bPass4															:= P_U01.vacuum_pump_inlet_valve_clear;
		bPass5															:= P_U01.vacuum_pump_bypass_valve_clear;
		IF rs_valves_clear AND bPass1 AND bPass2 AND bPass3 AND bPass4 AND bPass5 THEN
			bTimer1														:= FALSE;
			IF P_U01.boiler_ready THEN																						// 2
				P_U01.condenser_fan										:= TRUE;
				P_U01.condenser_pump									:= TRUE;
				P_U01.steam_flow_control_valve_mode						:= eManual;											// 3
				P_U01.steam_flow_control_valve							:= _OPEN;
				steam_bypass_valve										:= TRUE;
				rTime1													:= _VALVE_TIME;
				i8Step													:= i8Step + 1;
			ELSE
				sUtilityError											:= gsBoilerError;
			END_IF
		ELSIF tonTimer1.Q THEN
			bTimer1														:= FALSE;
			sReactorError												:= SEL(dead_air_valve_clear, gsDeadAirValveError, '');
			sReactorError												:= SEL(product_iso_valve_clear, gsProductIsoValveError, sReactorError);
			sReactorError												:= SEL(condensate_valve_clear, gsCondensateValveError, sReactorError);
			sReactorError												:= SEL(steam_iso_valve_clear, gsSteamIsoValveError, sReactorError);
			sReactorError												:= SEL(steam_bypass_valve_clear, gsSteamBypassValveError, sReactorError);
			sUtilityError												:= SEL(bPass1, gsVacuumPressureControlValveError, '');
			sUtilityError												:= SEL(bPass2, gsSteamFlowConrolValveError, sUtilityError);
			sUtilityError												:= SEL(bPass3, gsProductLineAmbientValveError, sUtilityError);
			sUtilityError												:= SEL(bPass4, gsVacuumPumpInletValveError, sUtilityError);
			sUtilityError												:= SEL(bPass5, gsVacuumPumpBypassValveError, sUtilityError);
		END_IF
		
	4:
		bTimer1															:= TRUE;
		bPass1															:= P_U01.steam_flow_control_valve_open;
		bPass2															:= steam_bypass_valve_clear;
		IF bPass1 AND bPass2 THEN
			bTimer1														:= FALSE;
			cycle_stage													:= 'bypass.running';
			rTime1														:= P_U01.SP_minimum_steam_bypass_duration * _MINUTES;
			i8Step														:= i8Step + 1;
		ELSIF tonTimer1.Q THEN
			bTimer1														:= FALSE;
			sUtilityError												:= SEL(bPass1, gsSteamFlowConrolValveError, '');
			sReactorError												:= SEL(bPass2, gsSteamBypassValveError, '');
		END_IF
		
	5:	bTimer1															:= TRUE;
		IF tonTimer1.Q THEN
			bTimer1														:= FALSE;
			bPass1														:= P_U01.steam_flow > P_U01.SP_minimum_steam_bypass_flow_rate;
			bPass2														:= product_line_temp > 90;
			IF bPass1 AND bPass2 THEN
				steam_bypass_valve										:= FALSE;											// 4
				P_U01.steam_flow_control_valve_mode						:= eManual;											///@@@ Not specified in narrative
				P_U01.steam_flow_control_valve							:= _CLOSED;
				rTime1													:= _VALVE_TIME;										// 5
				i8Step													:= i8Step + 1;
			ELSE
				sUtilityError											:= SEL(bPass1, gsSteamFlowTooLowError, '');
				sReactorError											:= SEL(bPass2, gsProductLineTempTooLowError, '');
			END_IF
		END_IF

	6:
		bTimer1															:= TRUE;
		bPass1															:= P_U01.steam_flow_control_valve_closed;
		bPass2															:= steam_bypass_valve_clear;
		IF bPass1 AND bPass2 THEN
			bTimer1														:= FALSE;
			P_U01.vacuum_pump_bypass_valve								:= FALSE;											// 6
			P_U01.product_line_ambient_valve							:= TRUE;
			rTime1														:= _VALVE_TIME;
			i8Step														:= i8Step + 1;
		ELSIF tonTimer1.Q THEN
			bTimer1														:= FALSE;
			sUtilityError												:= SEL(bPass1, gsSteamFlowConrolValveError, '');
			sReactorError												:= SEL(bPass2, gsSteamBypassValveError, '');
		END_IF

	7:
		bTimer1															:= TRUE;
		bPass1															:= P_U01.product_line_ambient_valve_clear;
		bPass2															:= P_U01.vacuum_pump_bypass_valve_clear;
		IF bPass1 AND bPass2 THEN
			bTimer1														:= FALSE;
			i8Step														:= 99;
		ELSIF tonTimer1.Q THEN
			bTimer1														:= FALSE;
			sUtilityError												:= SEL(bPass1, gsProductLineAmbientValveError, '');
			sUtilityError												:= SEL(bPass2, gsVacuumPumpBypassValveError, sUtilityError);
		END_IF
		
	80:																														// Stop process
		cycle_stage														:= 'bypass.stopping';
		A_Reset();
		P_U01.drainage_on												:= FALSE;
		P_U01.vacuum_pump_bypass_valve									:= FALSE;
		P_U01.condenser_fan												:= FALSE;
		P_U01.condenser_pump											:= FALSE;
		P_U01.steam_flow_control_valve_mode								:= eManual;
		P_U01.steam_flow_control_valve									:= _CLOSED;
		P_U01.product_line_ambient_valve								:= FALSE;											///@@@ Correct position???
		rTime1															:= _STOPPING_TIME;
		i8Step															:= 98;
		
	90:																														// Automatic process stopping
		cycle_stage														:= 'bypass.stopping';
		A_Reset();
		rTime1															:= _STOPPING_TIME;
		i8Step															:= 98;
		
	98:
		bTimer1															:= TRUE;
		IF tonTimer1.Q THEN
			bTimer1														:= FALSE;
			i8Step														:= 99;
		END_IF
		
	99:
		bBypassDone														:= TRUE;											// 13
		Current_Step													:= 0;
		i8Step															:= 0;
	
